  PROC DrawPart209()
    MoveL Offs(pOrigin,365.71,175.16,0.00),v40,z0,tPen\WObj:=wPaper;
    MoveL Offs(pOrigin,365.26,175.89,0.00),v40,z0,tPen\WObj:=wPaper;
    MoveL Offs(pOrigin,362.26,172.89,0.00),v40,z0,tPen\WObj:=wPaper;
    MoveL Offs(pOrigin,361.82,173.07,0.00),v40,z0,tPen\WObj:=wPaper;
    MoveL Offs(pOrigin,364.22,170.67,0.00),v40,z0,tPen\WObj:=wPaper;
    MoveL Offs(pOrigin,364.05,171.69,0.00),v40,z0,tPen\WObj:=wPaper;
    MoveL Offs(pOrigin,360.89,168.54,0.00),v40,z0,tPen\WObj:=wPaper;
    MoveL Offs(pOrigin,360.63,168.28,0.00),v40,z0,tPen\WObj:=wPaper;
    MoveL Offs(pOrigin,363.04,165.88,0.00),v40,z0,tPen\WObj:=wPaper;
    MoveL Offs(pOrigin,362.23,165.40,0.00),v40,z0,tPen\WObj:=wPaper;
    MoveL Offs(pOrigin,359.38,162.54,0.00),v40,z0,tPen\WObj:=wPaper;
    MoveL Offs(pOrigin,358.85,162.59,0.00),v40,z0,tPen\WObj:=wPaper;
    MoveL Offs(pOrigin,361.26,160.19,0.00),v40,z0,tPen\WObj:=wPaper;
    MoveL Offs(pOrigin,361.70,161.24,0.00),v40,z0,tPen\WObj:=wPaper;
    MoveL Offs(pOrigin,359.30,163.64,0.00),v40,z0,tPen\WObj:=wPaper;
    MoveL Offs(pOrigin,360.08,162.84,0.00),v40,z0,tPen\WObj:=wPaper;
    MoveL Offs(pOrigin,361.14,162.84,0.00),v40,z0,tPen\WObj:=wPaper;
    MoveL Offs(pOrigin,361.85,162.59,0.00),v40,z0,tPen\WObj:=wPaper;
    MoveL Offs(pOrigin,359.60,164.84,0.00),v40,z0,tPen\WObj:=wPaper;
    MoveL Offs(pOrigin,359.98,164.64,0.00),v40,z0,tPen\WObj:=wPaper;
    MoveL Offs(pOrigin,362.84,167.49,0.00),v40,z0,tPen\WObj:=wPaper;
    MoveL Offs(pOrigin,363.18,167.23,0.00),v40,z0,tPen\WObj:=wPaper;
    MoveL Offs(pOrigin,360.78,169.63,0.00),v40,z0,tPen\WObj:=wPaper;
    MoveL Offs(pOrigin,361.23,170.68,0.00),v40,z0,tPen\WObj:=wPaper;
    MoveL Offs(pOrigin,363.63,168.27,0.00),v40,fine,tPen\WObj:=wPaper;
    MoveL Offs(pOrigin,363.63,168.27,6.00),v60,z5,tPen\WObj:=wPaper;
    MoveL Offs(pOrigin,360.19,167.23,6.00),vTravel,z5,tPen\WObj:=wPaper;
    MoveL Offs(pOrigin,360.19,167.23,0.00),v60,z0,tPen\WObj:=wPaper;
    MoveL Offs(pOrigin,362.59,164.83,0.00),v40,fine,tPen\WObj:=wPaper;
    MoveL Offs(pOrigin,362.59,164.83,6.00),v60,z5,tPen\WObj:=wPaper;
    MoveL Offs(pOrigin,361.17,161.35,6.00),vTravel,z5,tPen\WObj:=wPaper;
    MoveL Offs(pOrigin,361.17,161.35,0.00),v60,z0,tPen\WObj:=wPaper;
    MoveL Offs(pOrigin,358.32,158.49,0.00),v40,z0,tPen\WObj:=wPaper;
    MoveL Offs(pOrigin,357.97,159.00,0.00),v40,z0,tPen\WObj:=wPaper;
    MoveL Offs(pOrigin,360.52,156.45,0.00),v40,fine,tPen\WObj:=wPaper;
    MoveL Offs(pOrigin,360.52,156.45,6.00),v60,z5,tPen\WObj:=wPaper;
    MoveL Offs(pOrigin,360.67,157.80,6.00),vTravel,z5,tPen\WObj:=wPaper;
    MoveL Offs(pOrigin,360.67,157.80,0.00),v60,z0,tPen\WObj:=wPaper;
    MoveL Offs(pOrigin,358.26,160.20,0.00),v40,fine,tPen\WObj:=wPaper;
    MoveL Offs(pOrigin,358.26,160.20,6.00),v60,z5,tPen\WObj:=wPaper;
    MoveL Offs(pOrigin,358.56,161.40,6.00),vTravel,z5,tPen\WObj:=wPaper;
    MoveL Offs(pOrigin,358.56,161.40,0.00),v60,z0,tPen\WObj:=wPaper;
    MoveL Offs(pOrigin,361.11,158.84,0.00),v40,fine,tPen\WObj:=wPaper;
    MoveL Offs(pOrigin,361.11,158.84,6.00),v60,z5,tPen\WObj:=wPaper;
    MoveL Offs(pOrigin,365.31,157.63,6.00),vTravel,z5,tPen\WObj:=wPaper;
    MoveL Offs(pOrigin,365.31,157.63,0.00),v60,z0,tPen\WObj:=wPaper;
    MoveL Offs(pOrigin,366.81,156.13,0.00),v40,z0,tPen\WObj:=wPaper;
    MoveL Offs(pOrigin,366.22,155.23,0.00),v40,z0,tPen\WObj:=wPaper;
    MoveL Offs(pOrigin,364.86,156.58,0.00),v40,z0,tPen\WObj:=wPaper;
    MoveL Offs(pOrigin,364.27,155.69,0.00),v40,z0,tPen\WObj:=wPaper;
    MoveL Offs(pOrigin,365.62,154.33,0.00),v40,z0,tPen\WObj:=wPaper;
    MoveL Offs(pOrigin,364.96,155.02,0.00),v40,z0,tPen\WObj:=wPaper;
    MoveL Offs(pOrigin,365.17,155.45,0.00),v40,z0,tPen\WObj:=wPaper;
    MoveL Offs(pOrigin,364.96,155.02,0.00),v40,fine,tPen\WObj:=wPaper;
    MoveL Offs(pOrigin,364.96,155.02,6.00),v60,z5,tPen\WObj:=wPaper;
    MoveL Offs(pOrigin,363.82,154.64,6.00),vTravel,z5,tPen\WObj:=wPaper;
    MoveL Offs(pOrigin,363.82,154.64,0.00),v60,z0,tPen\WObj:=wPaper;
    MoveL Offs(pOrigin,365.17,153.29,0.00),v40,z0,tPen\WObj:=wPaper;
    MoveL Offs(pOrigin,364.43,152.54,0.00),v40,z0,tPen\WObj:=wPaper;
    MoveL Offs(pOrigin,363.38,153.59,0.00),v40,z0,tPen\WObj:=wPaper;
    MoveL Offs(pOrigin,362.93,152.55,0.00),v40,z0,tPen\WObj:=wPaper;
    MoveL Offs(pOrigin,363.83,151.64,0.00),v40,fine,tPen\WObj:=wPaper;
    MoveL Offs(pOrigin,363.83,151.64,6.00),v60,z5,tPen\WObj:=wPaper;
    MoveL Offs(pOrigin,361.99,148.86,6.00),vTravel,z5,tPen\WObj:=wPaper;
    MoveL Offs(pOrigin,361.99,148.86,0.00),v60,z0,tPen\WObj:=wPaper;
    MoveL Offs(pOrigin,368.29,160.98,0.00),v40,z0,tPen\WObj:=wPaper;
    MoveL Offs(pOrigin,376.86,174.36,0.00),v40,z0,tPen\WObj:=wPaper;
    MoveL Offs(pOrigin,377.69,175.12,0.00),v40,z0,tPen\WObj:=wPaper;
    MoveL Offs(pOrigin,382.35,170.46,0.00),v40,fine,tPen\WObj:=wPaper;
    MoveL Offs(pOrigin,382.35,170.46,6.00),v60,z5,tPen\WObj:=wPaper;
    MoveL Offs(pOrigin,382.34,171.96,6.00),vTravel,z5,tPen\WObj:=wPaper;
    MoveL Offs(pOrigin,382.34,171.96,0.00),v60,z0,tPen\WObj:=wPaper;
    MoveL Offs(pOrigin,377.24,177.07,0.00),v40,fine,tPen\WObj:=wPaper;
    MoveL Offs(pOrigin,377.24,177.07,6.00),v60,z5,tPen\WObj:=wPaper;
    MoveL Offs(pOrigin,376.78,179.02,6.00),vTravel,z5,tPen\WObj:=wPaper;
    MoveL Offs(pOrigin,376.78,179.02,0.00),v60,z0,tPen\WObj:=wPaper;
    MoveL Offs(pOrigin,381.74,174.06,0.00),v40,fine,tPen\WObj:=wPaper;
    MoveL Offs(pOrigin,381.74,174.06,6.00),v60,z5,tPen\WObj:=wPaper;
    MoveL Offs(pOrigin,378.75,172.57,6.00),vTravel,z5,tPen\WObj:=wPaper;
    MoveL Offs(pOrigin,378.75,172.57,0.00),v60,z0,tPen\WObj:=wPaper;
    MoveL Offs(pOrigin,382.35,168.96,0.00),v40,fine,tPen\WObj:=wPaper;
    MoveL Offs(pOrigin,382.35,168.96,6.00),v60,z5,tPen\WObj:=wPaper;
    MoveL Offs(pOrigin,380.69,164.95,6.00),vTravel,z5,tPen\WObj:=wPaper;
    MoveL Offs(pOrigin,380.69,164.95,0.00),v60,z0,tPen\WObj:=wPaper;
    MoveL Offs(pOrigin,377.92,164.95,0.00),v40,z0,tPen\WObj:=wPaper;
    MoveL Offs(pOrigin,376.97,165.39,0.00),v40,z0,tPen\WObj:=wPaper;
    MoveL Offs(pOrigin,384.03,158.32,0.00),v40,fine,tPen\WObj:=wPaper;
    MoveL Offs(pOrigin,384.03,158.32,6.00),v60,z5,tPen\WObj:=wPaper;
    MoveL Offs(pOrigin,385.24,155.62,6.00),vTravel,z5,tPen\WObj:=wPaper;
    MoveL Offs(pOrigin,385.24,155.62,0.00),v60,z0,tPen\WObj:=wPaper;
    MoveL Offs(pOrigin,376.38,164.49,0.00),v40,z0,tPen\WObj:=wPaper;
    MoveL Offs(pOrigin,376.86,163.95,0.00),v40,z0,tPen\WObj:=wPaper;
    MoveL Offs(pOrigin,377.29,164.38,0.00),v40,z0,tPen\WObj:=wPaper;
    MoveL Offs(pOrigin,376.86,163.95,0.00),v40,z0,tPen\WObj:=wPaper;
    MoveL Offs(pOrigin,376.23,163.10,0.00),v40,z0,tPen\WObj:=wPaper;
    MoveL Offs(pOrigin,376.65,163.52,0.00),v40,z0,tPen\WObj:=wPaper;
    MoveL Offs(pOrigin,376.23,163.10,0.00),v40,fine,tPen\WObj:=wPaper;
    MoveL Offs(pOrigin,376.23,163.10,6.00),v60,z5,tPen\WObj:=wPaper;
    MoveL Offs(pOrigin,372.33,165.55,6.00),vTravel,z5,tPen\WObj:=wPaper;
    MoveL Offs(pOrigin,372.33,165.55,0.00),v60,z0,tPen\WObj:=wPaper;
    MoveL Offs(pOrigin,370.67,167.20,0.00),v40,z0,tPen\WObj:=wPaper;
    MoveL Offs(pOrigin,371.42,167.95,0.00),v40,z0,tPen\WObj:=wPaper;
    MoveL Offs(pOrigin,372.77,166.60,0.00),v40,z0,tPen\WObj:=wPaper;
    MoveL Offs(pOrigin,373.52,167.34,0.00),v40,z0,tPen\WObj:=wPaper;
    MoveL Offs(pOrigin,372.02,168.85,0.00),v40,z0,tPen\WObj:=wPaper;
    MoveL Offs(pOrigin,372.61,169.74,0.00),v40,z0,tPen\WObj:=wPaper;
    MoveL Offs(pOrigin,373.97,168.39,0.00),v40,z0,tPen\WObj:=wPaper;
    MoveL Offs(pOrigin,374.56,169.29,0.00),v40,z0,tPen\WObj:=wPaper;
    MoveL Offs(pOrigin,373.21,170.64,0.00),v40,z0,tPen\WObj:=wPaper;
    MoveL Offs(pOrigin,373.96,171.39,0.00),v40,z0,tPen\WObj:=wPaper;
    MoveL Offs(pOrigin,375.16,170.18,0.00),v40,z0,tPen\WObj:=wPaper;
    MoveL Offs(pOrigin,375.76,171.08,0.00),v40,z0,tPen\WObj:=wPaper;
    MoveL Offs(pOrigin,374.55,172.28,0.00),v40,z0,tPen\WObj:=wPaper;
    MoveL Offs(pOrigin,375.30,173.03,0.00),v40,z0,tPen\WObj:=wPaper;
    MoveL Offs(pOrigin,376.20,172.13,0.00),v40,fine,tPen\WObj:=wPaper;
    MoveL Offs(pOrigin,376.20,172.13,6.00),v60,z5,tPen\WObj:=wPaper;
    MoveL Offs(pOrigin,373.67,169.69,6.00),vTravel,z5,tPen\WObj:=wPaper;
    MoveL Offs(pOrigin,373.67,169.69,0.00),v60,z0,tPen\WObj:=wPaper;
    MoveL Offs(pOrigin,374.10,170.32,0.00),v40,z0,tPen\WObj:=wPaper;
    MoveL Offs(pOrigin,373.67,169.69,0.00),v40,fine,tPen\WObj:=wPaper;
  ENDPROC

  PROC DrawPart210()
    MoveL Offs(pOrigin,373.67,169.69,6.00),v60,z5,tPen\WObj:=wPaper;
    MoveL Offs(pOrigin,371.82,166.02,6.00),vTravel,z5,tPen\WObj:=wPaper;
    MoveL Offs(pOrigin,371.82,166.02,0.00),v60,z0,tPen\WObj:=wPaper;
    MoveL Offs(pOrigin,369.12,163.32,0.00),v40,z0,tPen\WObj:=wPaper;
    MoveL Offs(pOrigin,368.44,163.46,0.00),v40,z0,tPen\WObj:=wPaper;
    MoveL Offs(pOrigin,370.24,161.66,0.00),v40,z0,tPen\WObj:=wPaper;
    MoveL Offs(pOrigin,369.86,162.57,0.00),v40,z0,tPen\WObj:=wPaper;
    MoveL Offs(pOrigin,367.46,160.17,0.00),v40,z0,tPen\WObj:=wPaper;
    MoveL Offs(pOrigin,366.95,160.47,0.00),v40,z0,tPen\WObj:=wPaper;
    MoveL Offs(pOrigin,368.45,158.97,0.00),v40,z0,tPen\WObj:=wPaper;
    MoveL Offs(pOrigin,367.86,158.07,0.00),v40,z0,tPen\WObj:=wPaper;
    MoveL Offs(pOrigin,366.35,159.58,0.00),v40,z0,tPen\WObj:=wPaper;
    MoveL Offs(pOrigin,365.91,158.53,0.00),v40,z0,tPen\WObj:=wPaper;
    MoveL Offs(pOrigin,367.26,157.18,0.00),v40,z0,tPen\WObj:=wPaper;
    MoveL Offs(pOrigin,366.45,157.79,0.00),v40,z0,tPen\WObj:=wPaper;
    MoveL Offs(pOrigin,366.66,158.21,0.00),v40,z0,tPen\WObj:=wPaper;
    MoveL Offs(pOrigin,366.45,157.79,0.00),v40,fine,tPen\WObj:=wPaper;
    MoveL Offs(pOrigin,366.45,157.79,6.00),v60,z5,tPen\WObj:=wPaper;
    MoveL Offs(pOrigin,368.90,160.02,6.00),vTravel,z5,tPen\WObj:=wPaper;
    MoveL Offs(pOrigin,368.90,160.02,0.00),v60,z0,tPen\WObj:=wPaper;
    MoveL Offs(pOrigin,367.40,161.52,0.00),v40,z0,tPen\WObj:=wPaper;
    MoveL Offs(pOrigin,367.99,162.42,0.00),v40,z0,tPen\WObj:=wPaper;
    MoveL Offs(pOrigin,369.50,160.91,0.00),v40,fine,tPen\WObj:=wPaper;
    MoveL Offs(pOrigin,369.50,160.91,6.00),v60,z5,tPen\WObj:=wPaper;
    MoveL Offs(pOrigin,370.69,162.71,6.00),vTravel,z5,tPen\WObj:=wPaper;
    MoveL Offs(pOrigin,370.69,162.71,0.00),v60,z0,tPen\WObj:=wPaper;
    MoveL Offs(pOrigin,369.04,164.36,0.00),v40,z0,tPen\WObj:=wPaper;
    MoveL Offs(pOrigin,369.48,165.41,0.00),v40,z0,tPen\WObj:=wPaper;
    MoveL Offs(pOrigin,371.28,163.60,0.00),v40,z0,tPen\WObj:=wPaper;
    MoveL Offs(pOrigin,371.73,164.65,0.00),v40,z0,tPen\WObj:=wPaper;
    MoveL Offs(pOrigin,370.23,166.15,0.00),v40,fine,tPen\WObj:=wPaper;
    MoveL Offs(pOrigin,370.23,166.15,6.00),v60,z5,tPen\WObj:=wPaper;
    MoveL Offs(pOrigin,365.85,176.50,6.00),vTravel,z5,tPen\WObj:=wPaper;
    MoveL Offs(pOrigin,365.85,176.50,0.00),v60,z0,tPen\WObj:=wPaper;
    MoveL Offs(pOrigin,363.75,178.61,0.00),v40,fine,tPen\WObj:=wPaper;
    MoveL Offs(pOrigin,363.75,178.61,6.00),v60,z5,tPen\WObj:=wPaper;
    MoveL Offs(pOrigin,364.64,180.70,6.00),vTravel,z5,tPen\WObj:=wPaper;
    MoveL Offs(pOrigin,364.64,180.70,0.00),v60,z0,tPen\WObj:=wPaper;
    MoveL Offs(pOrigin,366.74,178.60,0.00),v40,fine,tPen\WObj:=wPaper;
    MoveL Offs(pOrigin,366.74,178.60,6.00),v60,z5,tPen\WObj:=wPaper;
    MoveL Offs(pOrigin,367.49,180.84,6.00),vTravel,z5,tPen\WObj:=wPaper;
    MoveL Offs(pOrigin,367.49,180.84,0.00),v60,z0,tPen\WObj:=wPaper;
    MoveL Offs(pOrigin,365.38,182.95,0.00),v40,z0,tPen\WObj:=wPaper;
    MoveL Offs(pOrigin,365.83,183.99,0.00),v40,z0,tPen\WObj:=wPaper;
    MoveL Offs(pOrigin,367.93,181.89,0.00),v40,fine,tPen\WObj:=wPaper;
    MoveL Offs(pOrigin,367.93,181.89,6.00),v60,z5,tPen\WObj:=wPaper;
    MoveL Offs(pOrigin,371.06,187.72,6.00),vTravel,z5,tPen\WObj:=wPaper;
    MoveL Offs(pOrigin,371.06,187.72,0.00),v60,z0,tPen\WObj:=wPaper;
    MoveL Offs(pOrigin,365.50,193.28,0.00),v40,z0,tPen\WObj:=wPaper;
    MoveL Offs(pOrigin,365.76,192.82,0.00),v40,z0,tPen\WObj:=wPaper;
    MoveL Offs(pOrigin,364.26,191.32,0.00),v40,fine,tPen\WObj:=wPaper;
    MoveL Offs(pOrigin,364.26,191.32,6.00),v60,z5,tPen\WObj:=wPaper;
    MoveL Offs(pOrigin,365.46,191.02,6.00),vTravel,z5,tPen\WObj:=wPaper;
    MoveL Offs(pOrigin,365.46,191.02,0.00),v60,z0,tPen\WObj:=wPaper;
    MoveL Offs(pOrigin,366.81,192.37,0.00),v40,z0,tPen\WObj:=wPaper;
    MoveL Offs(pOrigin,367.60,192.68,0.00),v40,z0,tPen\WObj:=wPaper;
    MoveL Offs(pOrigin,372.26,188.02,0.00),v40,z0,tPen\WObj:=wPaper;
    MoveL Offs(pOrigin,372.19,188.79,0.00),v40,z0,tPen\WObj:=wPaper;
    MoveL Offs(pOrigin,374.29,190.90,0.00),v40,z0,tPen\WObj:=wPaper;
    MoveL Offs(pOrigin,373.89,190.30,0.00),v40,z0,tPen\WObj:=wPaper;
    MoveL Offs(pOrigin,369.00,190.30,0.00),v40,z0,tPen\WObj:=wPaper;
    MoveL Offs(pOrigin,367.85,190.43,0.00),v40,z0,tPen\WObj:=wPaper;
    MoveL Offs(pOrigin,369.20,191.78,0.00),v40,z0,tPen\WObj:=wPaper;
    MoveL Offs(pOrigin,368.36,191.35,0.00),v40,z0,tPen\WObj:=wPaper;
    MoveL Offs(pOrigin,366.02,191.35,0.00),v40,z0,tPen\WObj:=wPaper;
    MoveL Offs(pOrigin,366.50,190.57,0.00),v40,z0,tPen\WObj:=wPaper;
    MoveL Offs(pOrigin,368.01,192.08,0.00),v40,fine,tPen\WObj:=wPaper;
    MoveL Offs(pOrigin,368.01,192.08,6.00),v60,z5,tPen\WObj:=wPaper;
    MoveL Offs(pOrigin,365.51,190.29,6.00),vTravel,z5,tPen\WObj:=wPaper;
    MoveL Offs(pOrigin,365.51,190.29,0.00),v60,z0,tPen\WObj:=wPaper;
    MoveL Offs(pOrigin,361.45,194.34,0.00),v40,z0,tPen\WObj:=wPaper;
    MoveL Offs(pOrigin,362.17,193.71,0.00),v40,z0,tPen\WObj:=wPaper;
    MoveL Offs(pOrigin,360.67,192.20,0.00),v40,z0,tPen\WObj:=wPaper;
    MoveL Offs(pOrigin,361.46,191.35,0.00),v40,z0,tPen\WObj:=wPaper;
    MoveL Offs(pOrigin,357.41,195.40,0.00),v40,z0,tPen\WObj:=wPaper;
    MoveL Offs(pOrigin,356.33,195.34,0.00),v40,z0,tPen\WObj:=wPaper;
    MoveL Offs(pOrigin,354.68,193.68,0.00),v40,fine,tPen\WObj:=wPaper;
    MoveL Offs(pOrigin,354.68,193.68,6.00),v60,z5,tPen\WObj:=wPaper;
    MoveL Offs(pOrigin,353.37,193.47,6.00),vTravel,z5,tPen\WObj:=wPaper;
    MoveL Offs(pOrigin,353.37,193.47,0.00),v60,z0,tPen\WObj:=wPaper;
    MoveL Offs(pOrigin,349.01,197.83,0.00),v40,fine,tPen\WObj:=wPaper;
    MoveL Offs(pOrigin,349.01,197.83,6.00),v60,z5,tPen\WObj:=wPaper;
    MoveL Offs(pOrigin,346.91,198.43,6.00),vTravel,z5,tPen\WObj:=wPaper;
    MoveL Offs(pOrigin,346.91,198.43,0.00),v60,z0,tPen\WObj:=wPaper;
    MoveL Offs(pOrigin,351.27,194.08,0.00),v40,z0,tPen\WObj:=wPaper;
    MoveL Offs(pOrigin,351.24,194.72,0.00),v40,z0,tPen\WObj:=wPaper;
    MoveL Offs(pOrigin,352.59,196.07,0.00),v40,z0,tPen\WObj:=wPaper;
    MoveL Offs(pOrigin,352.85,195.58,0.00),v40,z0,tPen\WObj:=wPaper;
    MoveL Offs(pOrigin,349.88,195.58,0.00),v40,z0,tPen\WObj:=wPaper;
    MoveL Offs(pOrigin,350.04,195.02,0.00),v40,z0,tPen\WObj:=wPaper;
    MoveL Offs(pOrigin,351.54,196.52,0.00),v40,fine,tPen\WObj:=wPaper;
    MoveL Offs(pOrigin,351.54,196.52,6.00),v60,z5,tPen\WObj:=wPaper;
    MoveL Offs(pOrigin,353.21,196.62,6.00),vTravel,z5,tPen\WObj:=wPaper;
    MoveL Offs(pOrigin,353.21,196.62,0.00),v60,z0,tPen\WObj:=wPaper;
    MoveL Offs(pOrigin,357.41,192.41,0.00),v40,z0,tPen\WObj:=wPaper;
    MoveL Offs(pOrigin,357.07,193.09,0.00),v40,z0,tPen\WObj:=wPaper;
    MoveL Offs(pOrigin,358.58,194.59,0.00),v40,fine,tPen\WObj:=wPaper;
    MoveL Offs(pOrigin,358.58,194.59,6.00),v60,z5,tPen\WObj:=wPaper;
    MoveL Offs(pOrigin,353.94,195.93,6.00),vTravel,z5,tPen\WObj:=wPaper;
    MoveL Offs(pOrigin,353.94,195.93,0.00),v60,z0,tPen\WObj:=wPaper;
    MoveL Offs(pOrigin,352.28,194.28,0.00),v40,fine,tPen\WObj:=wPaper;
    MoveL Offs(pOrigin,352.28,194.28,6.00),v60,z5,tPen\WObj:=wPaper;
    MoveL Offs(pOrigin,341.59,181.80,6.00),vTravel,z5,tPen\WObj:=wPaper;
    MoveL Offs(pOrigin,341.59,181.80,0.00),v60,z0,tPen\WObj:=wPaper;
    MoveL Offs(pOrigin,334.15,175.85,0.00),v40,z0,tPen\WObj:=wPaper;
    MoveL Offs(pOrigin,330.33,172.02,0.00),v40,z0,tPen\WObj:=wPaper;
    MoveL Offs(pOrigin,323.74,164.16,0.00),v40,z0,tPen\WObj:=wPaper;
    MoveL Offs(pOrigin,315.38,151.84,0.00),v40,z0,tPen\WObj:=wPaper;
    MoveL Offs(pOrigin,309.85,141.64,0.00),v40,z0,tPen\WObj:=wPaper;
    MoveL Offs(pOrigin,309.08,139.51,0.00),v40,fine,tPen\WObj:=wPaper;
    MoveL Offs(pOrigin,309.08,139.51,6.00),v60,z5,tPen\WObj:=wPaper;
    MoveL Offs(pOrigin,304.61,138.55,6.00),vTravel,z5,tPen\WObj:=wPaper;
    MoveL Offs(pOrigin,304.61,138.55,0.00),v60,z0,tPen\WObj:=wPaper;
    MoveL Offs(pOrigin,303.55,138.55,0.00),v40,z0,tPen\WObj:=wPaper;
    MoveL Offs(pOrigin,303.12,137.50,0.00),v40,z0,tPen\WObj:=wPaper;
    MoveL Offs(pOrigin,304.19,137.50,0.00),v40,z0,tPen\WObj:=wPaper;
    MoveL Offs(pOrigin,305.15,137.14,0.00),v40,z0,tPen\WObj:=wPaper;
    MoveL Offs(pOrigin,302.75,139.55,0.00),v40,fine,tPen\WObj:=wPaper;
    MoveL Offs(pOrigin,302.75,139.55,6.00),v60,z5,tPen\WObj:=wPaper;
    MoveL Offs(pOrigin,299.34,129.52,6.00),vTravel,z5,tPen\WObj:=wPaper;
  ENDPROC

  PROC DrawPart211()
    MoveL Offs(pOrigin,299.34,129.52,0.00),v60,z0,tPen\WObj:=wPaper;
    MoveL Offs(pOrigin,302.04,126.82,0.00),v40,fine,tPen\WObj:=wPaper;
    MoveL Offs(pOrigin,302.04,126.82,6.00),v60,z5,tPen\WObj:=wPaper;
    MoveL Offs(pOrigin,301.15,124.72,6.00),vTravel,z5,tPen\WObj:=wPaper;
    MoveL Offs(pOrigin,301.15,124.72,0.00),v60,z0,tPen\WObj:=wPaper;
    MoveL Offs(pOrigin,298.74,127.13,0.00),v40,fine,tPen\WObj:=wPaper;
    MoveL Offs(pOrigin,298.74,127.13,6.00),v60,z5,tPen\WObj:=wPaper;
    MoveL Offs(pOrigin,302.36,119.03,6.00),vTravel,z5,tPen\WObj:=wPaper;
    MoveL Offs(pOrigin,302.36,119.03,0.00),v60,z0,tPen\WObj:=wPaper;
    MoveL Offs(pOrigin,305.82,115.57,0.00),v40,z0,tPen\WObj:=wPaper;
    MoveL Offs(pOrigin,306.87,116.02,0.00),v40,z0,tPen\WObj:=wPaper;
    MoveL Offs(pOrigin,303.41,119.47,0.00),v40,z0,tPen\WObj:=wPaper;
    MoveL Offs(pOrigin,304.12,119.23,0.00),v40,z0,tPen\WObj:=wPaper;
    MoveL Offs(pOrigin,301.71,116.82,0.00),v40,fine,tPen\WObj:=wPaper;
    MoveL Offs(pOrigin,301.71,116.82,6.00),v60,z5,tPen\WObj:=wPaper;
    MoveL Offs(pOrigin,304.11,117.73,6.00),vTravel,z5,tPen\WObj:=wPaper;
    MoveL Offs(pOrigin,304.11,117.73,0.00),v60,z0,tPen\WObj:=wPaper;
    MoveL Offs(pOrigin,306.37,119.98,0.00),v40,z0,tPen\WObj:=wPaper;
    MoveL Offs(pOrigin,305.81,120.06,0.00),v40,z0,tPen\WObj:=wPaper;
    MoveL Offs(pOrigin,309.41,116.46,0.00),v40,z0,tPen\WObj:=wPaper;
    MoveL Offs(pOrigin,310.46,116.90,0.00),v40,z0,tPen\WObj:=wPaper;
    MoveL Offs(pOrigin,307.00,120.36,0.00),v40,z0,tPen\WObj:=wPaper;
    MoveL Offs(pOrigin,308.05,120.81,0.00),v40,z0,tPen\WObj:=wPaper;
    MoveL Offs(pOrigin,311.81,117.05,0.00),v40,fine,tPen\WObj:=wPaper;
    MoveL Offs(pOrigin,311.81,117.05,6.00),v60,z5,tPen\WObj:=wPaper;
    MoveL Offs(pOrigin,313.00,117.35,6.00),vTravel,z5,tPen\WObj:=wPaper;
    MoveL Offs(pOrigin,313.00,117.35,0.00),v60,z0,tPen\WObj:=wPaper;
    MoveL Offs(pOrigin,309.40,120.95,0.00),v40,z0,tPen\WObj:=wPaper;
    MoveL Offs(pOrigin,308.47,120.59,0.00),v40,z0,tPen\WObj:=wPaper;
    MoveL Offs(pOrigin,306.06,118.19,0.00),v40,fine,tPen\WObj:=wPaper;
    MoveL Offs(pOrigin,306.06,118.19,6.00),v60,z5,tPen\WObj:=wPaper;
    MoveL Offs(pOrigin,304.61,119.77,6.00),vTravel,z5,tPen\WObj:=wPaper;
    MoveL Offs(pOrigin,304.61,119.77,0.00),v60,z0,tPen\WObj:=wPaper;
    MoveL Offs(pOrigin,308.22,116.16,0.00),v40,fine,tPen\WObj:=wPaper;
    MoveL Offs(pOrigin,308.22,116.16,6.00),v60,z5,tPen\WObj:=wPaper;
    MoveL Offs(pOrigin,308.16,118.79,6.00),vTravel,z5,tPen\WObj:=wPaper;
    MoveL Offs(pOrigin,308.16,118.79,0.00),v60,z0,tPen\WObj:=wPaper;
    MoveL Offs(pOrigin,310.42,121.05,0.00),v40,z0,tPen\WObj:=wPaper;
    MoveL Offs(pOrigin,310.45,121.40,0.00),v40,z0,tPen\WObj:=wPaper;
    MoveL Offs(pOrigin,314.20,117.64,0.00),v40,fine,tPen\WObj:=wPaper;
    MoveL Offs(pOrigin,314.20,117.64,6.00),v60,z5,tPen\WObj:=wPaper;
    MoveL Offs(pOrigin,315.40,117.94,6.00),vTravel,z5,tPen\WObj:=wPaper;
    MoveL Offs(pOrigin,315.40,117.94,0.00),v60,z0,tPen\WObj:=wPaper;
    MoveL Offs(pOrigin,311.79,121.54,0.00),v40,z0,tPen\WObj:=wPaper;
    MoveL Offs(pOrigin,312.51,121.65,0.00),v40,z0,tPen\WObj:=wPaper;
    MoveL Offs(pOrigin,310.11,119.25,0.00),v40,fine,tPen\WObj:=wPaper;
    MoveL Offs(pOrigin,310.11,119.25,6.00),v60,z5,tPen\WObj:=wPaper;
    MoveL Offs(pOrigin,312.84,121.99,6.00),vTravel,z5,tPen\WObj:=wPaper;
    MoveL Offs(pOrigin,312.84,121.99,0.00),v60,z0,tPen\WObj:=wPaper;
    MoveL Offs(pOrigin,316.45,118.38,0.00),v40,fine,tPen\WObj:=wPaper;
    MoveL Offs(pOrigin,316.45,118.38,6.00),v60,z5,tPen\WObj:=wPaper;
    MoveL Offs(pOrigin,356.89,119.54,6.00),vTravel,z5,tPen\WObj:=wPaper;
    MoveL Offs(pOrigin,356.89,119.54,0.00),v60,z0,tPen\WObj:=wPaper;
    MoveL Offs(pOrigin,357.31,119.96,0.00),v40,z0,tPen\WObj:=wPaper;
    MoveL Offs(pOrigin,356.89,119.54,0.00),v40,fine,tPen\WObj:=wPaper;
    MoveL Offs(pOrigin,356.89,119.54,6.00),v60,z5,tPen\WObj:=wPaper;
    MoveL Offs(pOrigin,365.73,118.38,6.00),vTravel,z5,tPen\WObj:=wPaper;
    MoveL Offs(pOrigin,365.73,118.38,0.00),v60,z0,tPen\WObj:=wPaper;
    MoveL Offs(pOrigin,367.23,116.88,0.00),v40,z0,tPen\WObj:=wPaper;
    MoveL Offs(pOrigin,368.13,117.48,0.00),v40,z0,tPen\WObj:=wPaper;
    MoveL Offs(pOrigin,367.08,118.53,0.00),v40,fine,tPen\WObj:=wPaper;
    MoveL Offs(pOrigin,367.08,118.53,6.00),v60,z5,tPen\WObj:=wPaper;
    MoveL Offs(pOrigin,366.19,114.94,6.00),vTravel,z5,tPen\WObj:=wPaper;
    MoveL Offs(pOrigin,366.19,114.94,0.00),v60,z0,tPen\WObj:=wPaper;
    MoveL Offs(pOrigin,367.84,113.28,0.00),v40,fine,tPen\WObj:=wPaper;
    MoveL Offs(pOrigin,367.84,113.28,6.00),v60,z5,tPen\WObj:=wPaper;
    MoveL Offs(pOrigin,368.90,109.24,6.00),vTravel,z5,tPen\WObj:=wPaper;
    MoveL Offs(pOrigin,368.90,109.24,0.00),v60,z0,tPen\WObj:=wPaper;
    MoveL Offs(pOrigin,371.01,107.13,0.00),v40,z0,tPen\WObj:=wPaper;
    MoveL Offs(pOrigin,370.44,107.90,0.00),v40,z0,tPen\WObj:=wPaper;
    MoveL Offs(pOrigin,371.80,109.25,0.00),v40,z0,tPen\WObj:=wPaper;
    MoveL Offs(pOrigin,371.60,109.53,0.00),v40,z0,tPen\WObj:=wPaper;
    MoveL Offs(pOrigin,373.85,107.27,0.00),v40,z0,tPen\WObj:=wPaper;
    MoveL Offs(pOrigin,373.59,108.06,0.00),v40,z0,tPen\WObj:=wPaper;
    MoveL Offs(pOrigin,374.79,109.26,0.00),v40,z0,tPen\WObj:=wPaper;
    MoveL Offs(pOrigin,374.45,109.67,0.00),v40,z0,tPen\WObj:=wPaper;
    MoveL Offs(pOrigin,376.85,107.26,0.00),v40,fine,tPen\WObj:=wPaper;
    MoveL Offs(pOrigin,376.85,107.26,6.00),v60,z5,tPen\WObj:=wPaper;
    MoveL Offs(pOrigin,378.08,108.07,6.00),vTravel,z5,tPen\WObj:=wPaper;
    MoveL Offs(pOrigin,378.08,108.07,0.00),v60,z0,tPen\WObj:=wPaper;
    MoveL Offs(pOrigin,378.99,108.97,0.00),v40,z0,tPen\WObj:=wPaper;
    MoveL Offs(pOrigin,379.09,109.50,0.00),v40,z0,tPen\WObj:=wPaper;
    MoveL Offs(pOrigin,381.80,106.80,0.00),v40,fine,tPen\WObj:=wPaper;
    MoveL Offs(pOrigin,381.80,106.80,6.00),v60,z5,tPen\WObj:=wPaper;
    MoveL Offs(pOrigin,380.93,107.93,6.00),vTravel,z5,tPen\WObj:=wPaper;
    MoveL Offs(pOrigin,380.93,107.93,0.00),v60,z0,tPen\WObj:=wPaper;
    MoveL Offs(pOrigin,381.68,108.68,0.00),v40,z0,tPen\WObj:=wPaper;
    MoveL Offs(pOrigin,380.89,109.20,0.00),v40,z0,tPen\WObj:=wPaper;
    MoveL Offs(pOrigin,383.44,106.64,0.00),v40,fine,tPen\WObj:=wPaper;
    MoveL Offs(pOrigin,383.44,106.64,6.00),v60,z5,tPen\WObj:=wPaper;
    MoveL Offs(pOrigin,383.15,105.45,6.00),vTravel,z5,tPen\WObj:=wPaper;
    MoveL Offs(pOrigin,383.15,105.45,0.00),v60,z0,tPen\WObj:=wPaper;
    MoveL Offs(pOrigin,387.05,101.54,0.00),v40,z0,tPen\WObj:=wPaper;
    MoveL Offs(pOrigin,387.36,102.41,0.00),v40,z0,tPen\WObj:=wPaper;
    MoveL Offs(pOrigin,388.56,103.61,0.00),v40,z0,tPen\WObj:=wPaper;
    MoveL Offs(pOrigin,389.14,103.93,0.00),v40,z0,tPen\WObj:=wPaper;
    MoveL Offs(pOrigin,394.10,98.97,0.00),v40,z0,tPen\WObj:=wPaper;
    MoveL Offs(pOrigin,393.94,100.03,0.00),v40,z0,tPen\WObj:=wPaper;
    MoveL Offs(pOrigin,394.99,101.08,0.00),v40,z0,tPen\WObj:=wPaper;
    MoveL Offs(pOrigin,393.94,101.53,0.00),v40,z0,tPen\WObj:=wPaper;
    MoveL Offs(pOrigin,392.74,100.33,0.00),v40,z0,tPen\WObj:=wPaper;
    MoveL Offs(pOrigin,393.44,100.84,0.00),v40,z0,tPen\WObj:=wPaper;
    MoveL Offs(pOrigin,384.51,103.39,0.00),v40,z0,tPen\WObj:=wPaper;
    MoveL Offs(pOrigin,379.20,104.24,0.00),v40,z0,tPen\WObj:=wPaper;
    MoveL Offs(pOrigin,371.55,104.24,0.00),v40,z0,tPen\WObj:=wPaper;
    MoveL Offs(pOrigin,365.39,102.75,0.00),v40,fine,tPen\WObj:=wPaper;
    MoveL Offs(pOrigin,365.39,102.75,6.00),v60,z5,tPen\WObj:=wPaper;
    MoveL Offs(pOrigin,366.07,104.60,6.00),vTravel,z5,tPen\WObj:=wPaper;
    MoveL Offs(pOrigin,366.07,104.60,0.00),v60,z0,tPen\WObj:=wPaper;
    MoveL Offs(pOrigin,368.18,102.50,0.00),v40,z0,tPen\WObj:=wPaper;
    MoveL Offs(pOrigin,368.93,103.40,0.00),v40,z0,tPen\WObj:=wPaper;
    MoveL Offs(pOrigin,370.89,105.35,0.00),v40,z0,tPen\WObj:=wPaper;
    MoveL Offs(pOrigin,371.01,105.63,0.00),v40,z0,tPen\WObj:=wPaper;
    MoveL Offs(pOrigin,373.42,103.23,0.00),v40,z0,tPen\WObj:=wPaper;
    MoveL Offs(pOrigin,374.03,104.01,0.00),v40,z0,tPen\WObj:=wPaper;
    MoveL Offs(pOrigin,375.83,105.82,0.00),v40,z0,tPen\WObj:=wPaper;
    MoveL Offs(pOrigin,375.06,106.07,0.00),v40,z0,tPen\WObj:=wPaper;
    MoveL Offs(pOrigin,377.91,103.22,0.00),v40,z0,tPen\WObj:=wPaper;
    MoveL Offs(pOrigin,378.37,103.88,0.00),v40,z0,tPen\WObj:=wPaper;
    MoveL Offs(pOrigin,379.87,105.38,0.00),v40,z0,tPen\WObj:=wPaper;
  ENDPROC

  PROC DrawPart212()
    MoveL Offs(pOrigin,379.70,105.91,0.00),v40,z0,tPen\WObj:=wPaper;
    MoveL Offs(pOrigin,383.01,102.60,0.00),v40,z0,tPen\WObj:=wPaper;
    MoveL Offs(pOrigin,383.76,103.29,0.00),v40,z0,tPen\WObj:=wPaper;
    MoveL Offs(pOrigin,385.12,104.65,0.00),v40,fine,tPen\WObj:=wPaper;
    MoveL Offs(pOrigin,385.12,104.65,6.00),v60,z5,tPen\WObj:=wPaper;
    MoveL Offs(pOrigin,383.77,104.79,6.00),vTravel,z5,tPen\WObj:=wPaper;
    MoveL Offs(pOrigin,383.77,104.79,0.00),v60,z0,tPen\WObj:=wPaper;
    MoveL Offs(pOrigin,382.41,103.44,0.00),v40,fine,tPen\WObj:=wPaper;
    MoveL Offs(pOrigin,382.41,103.44,6.00),v60,z5,tPen\WObj:=wPaper;
    MoveL Offs(pOrigin,381.22,103.74,6.00),vTravel,z5,tPen\WObj:=wPaper;
    MoveL Offs(pOrigin,381.22,103.74,0.00),v60,z0,tPen\WObj:=wPaper;
    MoveL Offs(pOrigin,382.57,105.09,0.00),v40,fine,tPen\WObj:=wPaper;
    MoveL Offs(pOrigin,382.57,105.09,6.00),v60,z5,tPen\WObj:=wPaper;
    MoveL Offs(pOrigin,381.36,102.76,6.00),vTravel,z5,tPen\WObj:=wPaper;
    MoveL Offs(pOrigin,381.36,102.76,0.00),v60,z0,tPen\WObj:=wPaper;
    MoveL Offs(pOrigin,378.05,106.06,0.00),v40,z0,tPen\WObj:=wPaper;
    MoveL Offs(pOrigin,378.68,105.68,0.00),v40,z0,tPen\WObj:=wPaper;
    MoveL Offs(pOrigin,377.02,104.02,0.00),v40,z0,tPen\WObj:=wPaper;
    MoveL Offs(pOrigin,377.29,104.76,0.00),v40,z0,tPen\WObj:=wPaper;
    MoveL Offs(pOrigin,373.67,104.76,0.00),v40,fine,tPen\WObj:=wPaper;
    MoveL Offs(pOrigin,373.67,104.76,6.00),v60,z5,tPen\WObj:=wPaper;
    MoveL Offs(pOrigin,374.33,105.81,6.00),vTravel,z5,tPen\WObj:=wPaper;
    MoveL Offs(pOrigin,374.33,105.81,0.00),v60,z0,tPen\WObj:=wPaper;
    MoveL Offs(pOrigin,372.38,103.86,0.00),v40,z0,tPen\WObj:=wPaper;
    MoveL Offs(pOrigin,371.92,103.23,0.00),v40,z0,tPen\WObj:=wPaper;
    MoveL Offs(pOrigin,369.67,105.49,0.00),v40,fine,tPen\WObj:=wPaper;
    MoveL Offs(pOrigin,369.67,105.49,6.00),v60,z5,tPen\WObj:=wPaper;
    MoveL Offs(pOrigin,369.51,107.14,6.00),vTravel,z5,tPen\WObj:=wPaper;
    MoveL Offs(pOrigin,369.51,107.14,0.00),v60,z0,tPen\WObj:=wPaper;
    MoveL Offs(pOrigin,367.56,109.09,0.00),v40,z0,tPen\WObj:=wPaper;
    MoveL Offs(pOrigin,368.20,108.64,0.00),v40,z0,tPen\WObj:=wPaper;
    MoveL Offs(pOrigin,367.15,107.59,0.00),v40,z0,tPen\WObj:=wPaper;
    MoveL Offs(pOrigin,366.97,106.69,0.00),v40,z0,tPen\WObj:=wPaper;
    MoveL Offs(pOrigin,365.16,108.50,0.00),v40,z0,tPen\WObj:=wPaper;
    MoveL Offs(pOrigin,364.12,108.05,0.00),v40,z0,tPen\WObj:=wPaper;
    MoveL Offs(pOrigin,365.77,106.40,0.00),v40,fine,tPen\WObj:=wPaper;
    MoveL Offs(pOrigin,365.77,106.40,6.00),v60,z5,tPen\WObj:=wPaper;
    MoveL Offs(pOrigin,364.42,106.25,6.00),vTravel,z5,tPen\WObj:=wPaper;
    MoveL Offs(pOrigin,364.42,106.25,0.00),v60,z0,tPen\WObj:=wPaper;
    MoveL Offs(pOrigin,362.92,107.76,0.00),v40,z0,tPen\WObj:=wPaper;
    MoveL Offs(pOrigin,361.87,107.31,0.00),v40,z0,tPen\WObj:=wPaper;
    MoveL Offs(pOrigin,363.37,105.81,0.00),v40,fine,tPen\WObj:=wPaper;
    MoveL Offs(pOrigin,363.37,105.81,6.00),v60,z5,tPen\WObj:=wPaper;
    MoveL Offs(pOrigin,362.18,105.51,6.00),vTravel,z5,tPen\WObj:=wPaper;
    MoveL Offs(pOrigin,362.18,105.51,0.00),v60,z0,tPen\WObj:=wPaper;
    MoveL Offs(pOrigin,360.82,106.86,0.00),v40,z0,tPen\WObj:=wPaper;
    MoveL Offs(pOrigin,359.93,106.27,0.00),v40,z0,tPen\WObj:=wPaper;
    MoveL Offs(pOrigin,360.98,105.21,0.00),v40,z0,tPen\WObj:=wPaper;
    MoveL Offs(pOrigin,359.93,104.77,0.00),v40,z0,tPen\WObj:=wPaper;
    MoveL Offs(pOrigin,358.73,105.97,0.00),v40,fine,tPen\WObj:=wPaper;
    MoveL Offs(pOrigin,358.73,105.97,6.00),v60,z5,tPen\WObj:=wPaper;
    MoveL Offs(pOrigin,357.52,107.93,6.00),vTravel,z5,tPen\WObj:=wPaper;
    MoveL Offs(pOrigin,357.52,107.93,0.00),v60,z0,tPen\WObj:=wPaper;
    MoveL Offs(pOrigin,356.46,107.93,0.00),v40,fine,tPen\WObj:=wPaper;
    MoveL Offs(pOrigin,356.46,107.93,6.00),v60,z5,tPen\WObj:=wPaper;
    MoveL Offs(pOrigin,362.33,102.36,6.00),vTravel,z5,tPen\WObj:=wPaper;
    MoveL Offs(pOrigin,362.33,102.36,0.00),v60,z0,tPen\WObj:=wPaper;
    MoveL Offs(pOrigin,363.99,100.71,0.00),v40,z0,tPen\WObj:=wPaper;
    MoveL Offs(pOrigin,363.83,101.29,0.00),v40,z0,tPen\WObj:=wPaper;
    MoveL Offs(pOrigin,367.14,104.59,0.00),v40,z0,tPen\WObj:=wPaper;
    MoveL Offs(pOrigin,367.27,104.90,0.00),v40,z0,tPen\WObj:=wPaper;
    MoveL Offs(pOrigin,369.37,102.79,0.00),v40,fine,tPen\WObj:=wPaper;
    MoveL Offs(pOrigin,369.37,102.79,6.00),v60,z5,tPen\WObj:=wPaper;
    MoveL Offs(pOrigin,368.31,106.84,6.00),vTravel,z5,tPen\WObj:=wPaper;
    MoveL Offs(pOrigin,368.31,106.84,0.00),v60,z0,tPen\WObj:=wPaper;
    MoveL Offs(pOrigin,366.51,108.64,0.00),v40,fine,tPen\WObj:=wPaper;
    MoveL Offs(pOrigin,366.51,108.64,6.00),v60,z5,tPen\WObj:=wPaper;
    MoveL Offs(pOrigin,368.95,107.89,6.00),vTravel,z5,tPen\WObj:=wPaper;
    MoveL Offs(pOrigin,368.95,107.89,0.00),v60,z0,tPen\WObj:=wPaper;
    MoveL Offs(pOrigin,370.00,108.94,0.00),v40,z0,tPen\WObj:=wPaper;
    MoveL Offs(pOrigin,370.10,109.53,0.00),v40,z0,tPen\WObj:=wPaper;
    MoveL Offs(pOrigin,372.36,107.28,0.00),v40,z0,tPen\WObj:=wPaper;
    MoveL Offs(pOrigin,372.09,108.05,0.00),v40,z0,tPen\WObj:=wPaper;
    MoveL Offs(pOrigin,373.30,109.25,0.00),v40,z0,tPen\WObj:=wPaper;
    MoveL Offs(pOrigin,372.95,109.67,0.00),v40,z0,tPen\WObj:=wPaper;
    MoveL Offs(pOrigin,375.35,107.27,0.00),v40,z0,tPen\WObj:=wPaper;
    MoveL Offs(pOrigin,375.39,108.36,0.00),v40,z0,tPen\WObj:=wPaper;
    MoveL Offs(pOrigin,376.14,109.11,0.00),v40,z0,tPen\WObj:=wPaper;
    MoveL Offs(pOrigin,375.94,109.66,0.00),v40,z0,tPen\WObj:=wPaper;
    MoveL Offs(pOrigin,378.35,107.26,0.00),v40,fine,tPen\WObj:=wPaper;
    MoveL Offs(pOrigin,378.35,107.26,6.00),v60,z5,tPen\WObj:=wPaper;
    MoveL Offs(pOrigin,379.58,108.08,6.00),vTravel,z5,tPen\WObj:=wPaper;
    MoveL Offs(pOrigin,379.58,108.08,0.00),v60,z0,tPen\WObj:=wPaper;
    MoveL Offs(pOrigin,380.33,108.83,0.00),v40,fine,tPen\WObj:=wPaper;
    MoveL Offs(pOrigin,380.33,108.83,6.00),v60,z5,tPen\WObj:=wPaper;
    MoveL Offs(pOrigin,380.00,107.10,6.00),vTravel,z5,tPen\WObj:=wPaper;
    MoveL Offs(pOrigin,380.00,107.10,0.00),v60,z0,tPen\WObj:=wPaper;
    MoveL Offs(pOrigin,377.44,109.66,0.00),v40,fine,tPen\WObj:=wPaper;
    MoveL Offs(pOrigin,377.44,109.66,6.00),v60,z5,tPen\WObj:=wPaper;
    MoveL Offs(pOrigin,373.56,106.08,6.00),vTravel,z5,tPen\WObj:=wPaper;
    MoveL Offs(pOrigin,373.56,106.08,0.00),v60,z0,tPen\WObj:=wPaper;
    MoveL Offs(pOrigin,376.41,103.22,0.00),v40,fine,tPen\WObj:=wPaper;
    MoveL Offs(pOrigin,376.41,103.22,6.00),v60,z5,tPen\WObj:=wPaper;
    MoveL Offs(pOrigin,371.98,108.70,6.00),vTravel,z5,tPen\WObj:=wPaper;
    MoveL Offs(pOrigin,371.98,108.70,0.00),v60,z0,tPen\WObj:=wPaper;
    MoveL Offs(pOrigin,371.55,108.06,0.00),v40,z0,tPen\WObj:=wPaper;
    MoveL Offs(pOrigin,370.91,108.06,0.00),v40,z0,tPen\WObj:=wPaper;
    MoveL Offs(pOrigin,370.70,108.49,0.00),v40,fine,tPen\WObj:=wPaper;
    MoveL Offs(pOrigin,370.70,108.49,6.00),v60,z5,tPen\WObj:=wPaper;
    MoveL Offs(pOrigin,375.77,117.30,6.00),vTravel,z5,tPen\WObj:=wPaper;
    MoveL Offs(pOrigin,375.77,117.30,0.00),v60,z0,tPen\WObj:=wPaper;
    MoveL Offs(pOrigin,374.12,118.96,0.00),v40,z0,tPen\WObj:=wPaper;
    MoveL Offs(pOrigin,375.02,119.55,0.00),v40,z0,tPen\WObj:=wPaper;
    MoveL Offs(pOrigin,376.82,117.75,0.00),v40,z0,tPen\WObj:=wPaper;
    MoveL Offs(pOrigin,376.32,118.25,0.00),v40,z0,tPen\WObj:=wPaper;
    MoveL Offs(pOrigin,378.57,120.51,0.00),v40,z0,tPen\WObj:=wPaper;
    MoveL Offs(pOrigin,379.20,121.34,0.00),v40,z0,tPen\WObj:=wPaper;
    MoveL Offs(pOrigin,380.86,119.68,0.00),v40,z0,tPen\WObj:=wPaper;
    MoveL Offs(pOrigin,381.90,120.13,0.00),v40,z0,tPen\WObj:=wPaper;
    MoveL Offs(pOrigin,380.25,121.78,0.00),v40,fine,tPen\WObj:=wPaper;
    MoveL Offs(pOrigin,380.25,121.78,6.00),v60,z5,tPen\WObj:=wPaper;
    MoveL Offs(pOrigin,381.14,123.88,6.00),vTravel,z5,tPen\WObj:=wPaper;
    MoveL Offs(pOrigin,381.14,123.88,0.00),v60,z0,tPen\WObj:=wPaper;
    MoveL Offs(pOrigin,379.79,125.23,0.00),v40,z0,tPen\WObj:=wPaper;
    MoveL Offs(pOrigin,378.99,124.64,0.00),v40,z0,tPen\WObj:=wPaper;
    MoveL Offs(pOrigin,384.51,125.70,0.00),v40,fine,tPen\WObj:=wPaper;
    MoveL Offs(pOrigin,384.51,125.70,6.00),v60,z5,tPen\WObj:=wPaper;
    MoveL Offs(pOrigin,385.94,123.56,6.00),vTravel,z5,tPen\WObj:=wPaper;
    MoveL Offs(pOrigin,385.94,123.56,0.00),v60,z0,tPen\WObj:=wPaper;
    MoveL Offs(pOrigin,386.84,122.66,0.00),v40,fine,tPen\WObj:=wPaper;
  ENDPROC

  PROC DrawPart213()
    MoveL Offs(pOrigin,386.84,122.66,6.00),v60,z5,tPen\WObj:=wPaper;
    MoveL Offs(pOrigin,383.85,121.17,6.00),vTravel,z5,tPen\WObj:=wPaper;
    MoveL Offs(pOrigin,383.85,121.17,0.00),v60,z0,tPen\WObj:=wPaper;
    MoveL Offs(pOrigin,382.35,122.68,0.00),v40,fine,tPen\WObj:=wPaper;
    MoveL Offs(pOrigin,382.35,122.68,6.00),v60,z5,tPen\WObj:=wPaper;
    MoveL Offs(pOrigin,382.34,124.17,6.00),vTravel,z5,tPen\WObj:=wPaper;
    MoveL Offs(pOrigin,382.34,124.17,0.00),v60,z0,tPen\WObj:=wPaper;
    MoveL Offs(pOrigin,380.84,125.68,0.00),v40,fine,tPen\WObj:=wPaper;
    MoveL Offs(pOrigin,380.84,125.68,6.00),v60,z5,tPen\WObj:=wPaper;
    MoveL Offs(pOrigin,387.72,127.75,6.00),vTravel,z5,tPen\WObj:=wPaper;
    MoveL Offs(pOrigin,387.72,127.75,0.00),v60,z0,tPen\WObj:=wPaper;
    MoveL Offs(pOrigin,389.83,125.65,0.00),v40,fine,tPen\WObj:=wPaper;
    MoveL Offs(pOrigin,389.83,125.65,6.00),v60,z5,tPen\WObj:=wPaper;
    MoveL Offs(pOrigin,391.17,125.79,6.00),vTravel,z5,tPen\WObj:=wPaper;
    MoveL Offs(pOrigin,391.17,125.79,0.00),v60,z0,tPen\WObj:=wPaper;
    MoveL Offs(pOrigin,388.62,128.35,0.00),v40,fine,tPen\WObj:=wPaper;
    MoveL Offs(pOrigin,388.62,128.35,6.00),v60,z5,tPen\WObj:=wPaper;
    MoveL Offs(pOrigin,389.61,130.10,6.00),vTravel,z5,tPen\WObj:=wPaper;
    MoveL Offs(pOrigin,389.61,130.10,0.00),v60,z0,tPen\WObj:=wPaper;
    MoveL Offs(pOrigin,391.10,130.10,0.00),v40,fine,tPen\WObj:=wPaper;
    MoveL Offs(pOrigin,391.10,130.10,6.00),v60,z5,tPen\WObj:=wPaper;
    MoveL Offs(pOrigin,392.85,128.89,6.00),vTravel,z5,tPen\WObj:=wPaper;
    MoveL Offs(pOrigin,392.85,128.89,0.00),v60,z0,tPen\WObj:=wPaper;
    MoveL Offs(pOrigin,392.85,127.61,0.00),v40,fine,tPen\WObj:=wPaper;
    MoveL Offs(pOrigin,392.85,127.61,6.00),v60,z5,tPen\WObj:=wPaper;
    MoveL Offs(pOrigin,394.71,126.34,6.00),vTravel,z5,tPen\WObj:=wPaper;
    MoveL Offs(pOrigin,394.71,126.34,0.00),v60,z0,tPen\WObj:=wPaper;
    MoveL Offs(pOrigin,394.50,126.76,0.00),v40,z0,tPen\WObj:=wPaper;
    MoveL Offs(pOrigin,394.71,126.34,0.00),v40,z0,tPen\WObj:=wPaper;
    MoveL Offs(pOrigin,395.14,125.88,0.00),v40,z0,tPen\WObj:=wPaper;
    MoveL Offs(pOrigin,396.41,125.88,0.00),v40,z0,tPen\WObj:=wPaper;
    MoveL Offs(pOrigin,396.62,124.82,0.00),v40,z0,tPen\WObj:=wPaper;
    MoveL Offs(pOrigin,395.56,124.82,0.00),v40,z0,tPen\WObj:=wPaper;
    MoveL Offs(pOrigin,395.56,123.77,0.00),v40,z0,tPen\WObj:=wPaper;
    MoveL Offs(pOrigin,396.62,123.77,0.00),v40,z0,tPen\WObj:=wPaper;
    MoveL Offs(pOrigin,396.62,122.71,0.00),v40,z0,tPen\WObj:=wPaper;
    MoveL Offs(pOrigin,395.56,122.71,0.00),v40,fine,tPen\WObj:=wPaper;
    MoveL Offs(pOrigin,395.56,122.71,6.00),v60,z5,tPen\WObj:=wPaper;
    MoveL Offs(pOrigin,397.63,122.33,6.00),vTravel,z5,tPen\WObj:=wPaper;
    MoveL Offs(pOrigin,397.63,122.33,0.00),v60,z0,tPen\WObj:=wPaper;
    MoveL Offs(pOrigin,388.46,131.50,0.00),v40,fine,tPen\WObj:=wPaper;
    MoveL Offs(pOrigin,388.46,131.50,6.00),v60,z5,tPen\WObj:=wPaper;
    MoveL Offs(pOrigin,392.16,135.38,6.00),vTravel,z5,tPen\WObj:=wPaper;
    MoveL Offs(pOrigin,392.16,135.38,0.00),v60,z0,tPen\WObj:=wPaper;
    MoveL Offs(pOrigin,393.44,135.38,0.00),v40,z0,tPen\WObj:=wPaper;
    MoveL Offs(pOrigin,393.22,136.44,0.00),v40,z0,tPen\WObj:=wPaper;
    MoveL Offs(pOrigin,392.16,136.44,0.00),v40,fine,tPen\WObj:=wPaper;
    MoveL Offs(pOrigin,392.16,136.44,6.00),v60,z5,tPen\WObj:=wPaper;
    MoveL Offs(pOrigin,393.82,141.07,6.00),vTravel,z5,tPen\WObj:=wPaper;
    MoveL Offs(pOrigin,393.82,141.07,0.00),v60,z0,tPen\WObj:=wPaper;
    MoveL Offs(pOrigin,390.07,144.82,0.00),v40,fine,tPen\WObj:=wPaper;
    MoveL Offs(pOrigin,390.07,144.82,6.00),v60,z5,tPen\WObj:=wPaper;
    MoveL Offs(pOrigin,389.91,147.97,6.00),vTravel,z5,tPen\WObj:=wPaper;
    MoveL Offs(pOrigin,389.91,147.97,0.00),v60,z0,tPen\WObj:=wPaper;
    MoveL Offs(pOrigin,393.36,144.51,0.00),v40,fine,tPen\WObj:=wPaper;
    MoveL Offs(pOrigin,393.36,144.51,6.00),v60,z5,tPen\WObj:=wPaper;
    MoveL Offs(pOrigin,391.74,151.22,6.00),vTravel,z5,tPen\WObj:=wPaper;
    MoveL Offs(pOrigin,391.74,151.22,0.00),v60,z0,tPen\WObj:=wPaper;
    MoveL Offs(pOrigin,390.67,151.22,0.00),v40,fine,tPen\WObj:=wPaper;
    MoveL Offs(pOrigin,390.67,151.22,6.00),v60,z5,tPen\WObj:=wPaper;
    MoveL Offs(pOrigin,392.13,156.20,6.00),vTravel,z5,tPen\WObj:=wPaper;
    MoveL Offs(pOrigin,392.13,156.20,0.00),v60,z0,tPen\WObj:=wPaper;
    MoveL Offs(pOrigin,388.67,159.66,0.00),v40,fine,tPen\WObj:=wPaper;
    MoveL Offs(pOrigin,388.67,159.66,6.00),v60,z5,tPen\WObj:=wPaper;
    MoveL Offs(pOrigin,389.83,160.73,6.00),vTravel,z5,tPen\WObj:=wPaper;
    MoveL Offs(pOrigin,389.83,160.73,0.00),v60,z0,tPen\WObj:=wPaper;
    MoveL Offs(pOrigin,390.89,160.73,0.00),v40,fine,tPen\WObj:=wPaper;
    MoveL Offs(pOrigin,390.89,160.73,6.00),v60,z5,tPen\WObj:=wPaper;
    MoveL Offs(pOrigin,391.66,162.64,6.00),vTravel,z5,tPen\WObj:=wPaper;
    MoveL Offs(pOrigin,391.66,162.64,0.00),v60,z0,tPen\WObj:=wPaper;
    MoveL Offs(pOrigin,388.20,166.10,0.00),v40,fine,tPen\WObj:=wPaper;
    MoveL Offs(pOrigin,388.20,166.10,6.00),v60,z5,tPen\WObj:=wPaper;
    MoveL Offs(pOrigin,389.40,164.95,6.00),vTravel,z5,tPen\WObj:=wPaper;
    MoveL Offs(pOrigin,389.40,164.95,0.00),v60,z0,tPen\WObj:=wPaper;
    MoveL Offs(pOrigin,390.46,164.95,0.00),v40,fine,tPen\WObj:=wPaper;
    MoveL Offs(pOrigin,390.46,164.95,6.00),v60,z5,tPen\WObj:=wPaper;
    MoveL Offs(pOrigin,390.89,169.39,6.00),vTravel,z5,tPen\WObj:=wPaper;
    MoveL Offs(pOrigin,390.89,169.39,0.00),v60,z0,tPen\WObj:=wPaper;
    MoveL Offs(pOrigin,387.58,172.69,0.00),v40,fine,tPen\WObj:=wPaper;
    MoveL Offs(pOrigin,387.58,172.69,6.00),v60,z5,tPen\WObj:=wPaper;
    MoveL Offs(pOrigin,388.76,171.29,6.00),vTravel,z5,tPen\WObj:=wPaper;
    MoveL Offs(pOrigin,388.76,171.29,0.00),v60,z0,tPen\WObj:=wPaper;
    MoveL Offs(pOrigin,389.83,171.29,0.00),v40,fine,tPen\WObj:=wPaper;
    MoveL Offs(pOrigin,389.83,171.29,6.00),v60,z5,tPen\WObj:=wPaper;
    MoveL Offs(pOrigin,390.43,174.33,6.00),vTravel,z5,tPen\WObj:=wPaper;
    MoveL Offs(pOrigin,390.43,174.33,0.00),v60,z0,tPen\WObj:=wPaper;
    MoveL Offs(pOrigin,387.12,177.64,0.00),v40,fine,tPen\WObj:=wPaper;
    MoveL Offs(pOrigin,387.12,177.64,6.00),v60,z5,tPen\WObj:=wPaper;
    MoveL Offs(pOrigin,387.59,178.81,6.00),vTravel,z5,tPen\WObj:=wPaper;
    MoveL Offs(pOrigin,387.59,178.81,0.00),v60,z0,tPen\WObj:=wPaper;
    MoveL Offs(pOrigin,389.39,180.61,0.00),v40,z0,tPen\WObj:=wPaper;
    MoveL Offs(pOrigin,389.81,180.92,0.00),v40,z0,tPen\WObj:=wPaper;
    MoveL Offs(pOrigin,386.50,184.23,0.00),v40,z0,tPen\WObj:=wPaper;
    MoveL Offs(pOrigin,387.16,184.35,0.00),v40,z0,tPen\WObj:=wPaper;
    MoveL Offs(pOrigin,388.81,186.00,0.00),v40,fine,tPen\WObj:=wPaper;
    MoveL Offs(pOrigin,388.81,186.00,6.00),v60,z5,tPen\WObj:=wPaper;
    MoveL Offs(pOrigin,388.34,187.13,6.00),vTravel,z5,tPen\WObj:=wPaper;
    MoveL Offs(pOrigin,388.34,187.13,0.00),v60,z0,tPen\WObj:=wPaper;
    MoveL Offs(pOrigin,387.28,187.13,0.00),v40,z0,tPen\WObj:=wPaper;
    MoveL Offs(pOrigin,386.87,187.04,0.00),v40,z0,tPen\WObj:=wPaper;
    MoveL Offs(pOrigin,388.52,188.69,0.00),v40,z0,tPen\WObj:=wPaper;
    MoveL Offs(pOrigin,388.12,189.24,0.00),v40,z0,tPen\WObj:=wPaper;
    MoveL Offs(pOrigin,387.06,189.24,0.00),v40,fine,tPen\WObj:=wPaper;
    MoveL Offs(pOrigin,387.06,189.24,6.00),v60,z5,tPen\WObj:=wPaper;
    MoveL Offs(pOrigin,389.18,189.02,6.00),vTravel,z5,tPen\WObj:=wPaper;
    MoveL Offs(pOrigin,389.18,189.02,0.00),v60,z0,tPen\WObj:=wPaper;
    MoveL Offs(pOrigin,385.58,192.62,0.00),v40,fine,tPen\WObj:=wPaper;
    MoveL Offs(pOrigin,385.58,192.62,6.00),v60,z5,tPen\WObj:=wPaper;
    MoveL Offs(pOrigin,385.85,196.48,6.00),vTravel,z5,tPen\WObj:=wPaper;
    MoveL Offs(pOrigin,385.85,196.48,0.00),v60,z0,tPen\WObj:=wPaper;
    MoveL Offs(pOrigin,387.65,198.28,0.00),v40,fine,tPen\WObj:=wPaper;
    MoveL Offs(pOrigin,387.65,198.28,6.00),v60,z5,tPen\WObj:=wPaper;
    MoveL Offs(pOrigin,381.51,198.18,6.00),vTravel,z5,tPen\WObj:=wPaper;
    MoveL Offs(pOrigin,381.51,198.18,0.00),v60,z0,tPen\WObj:=wPaper;
    MoveL Offs(pOrigin,379.11,200.58,0.00),v40,z0,tPen\WObj:=wPaper;
    MoveL Offs(pOrigin,379.42,200.50,0.00),v40,z0,tPen\WObj:=wPaper;
    MoveL Offs(pOrigin,381.52,202.60,0.00),v40,z0,tPen\WObj:=wPaper;
    MoveL Offs(pOrigin,381.80,202.37,0.00),v40,z0,tPen\WObj:=wPaper;
    MoveL Offs(pOrigin,379.25,204.93,0.00),v40,z0,tPen\WObj:=wPaper;
    MoveL Offs(pOrigin,379.88,205.45,0.00),v40,z0,tPen\WObj:=wPaper;
  ENDPROC

  PROC DrawPart214()
    MoveL Offs(pOrigin,381.68,207.25,0.00),v40,fine,tPen\WObj:=wPaper;
    MoveL Offs(pOrigin,381.68,207.25,6.00),v60,z5,tPen\WObj:=wPaper;
    MoveL Offs(pOrigin,379.39,206.27,6.00),vTravel,z5,tPen\WObj:=wPaper;
    MoveL Offs(pOrigin,379.39,206.27,0.00),v60,z0,tPen\WObj:=wPaper;
    MoveL Offs(pOrigin,382.10,203.57,0.00),v40,z0,tPen\WObj:=wPaper;
    MoveL Offs(pOrigin,381.53,204.10,0.00),v40,z0,tPen\WObj:=wPaper;
    MoveL Offs(pOrigin,379.72,202.30,0.00),v40,fine,tPen\WObj:=wPaper;
    MoveL Offs(pOrigin,379.72,202.30,6.00),v60,z5,tPen\WObj:=wPaper;
    MoveL Offs(pOrigin,376.57,200.14,6.00),vTravel,z5,tPen\WObj:=wPaper;
    MoveL Offs(pOrigin,376.57,200.14,0.00),v60,z0,tPen\WObj:=wPaper;
    MoveL Offs(pOrigin,374.16,202.54,0.00),v40,fine,tPen\WObj:=wPaper;
    MoveL Offs(pOrigin,374.16,202.54,6.00),v60,z5,tPen\WObj:=wPaper;
    MoveL Offs(pOrigin,373.57,200.15,6.00),vTravel,z5,tPen\WObj:=wPaper;
    MoveL Offs(pOrigin,373.57,200.15,0.00),v60,z0,tPen\WObj:=wPaper;
    MoveL Offs(pOrigin,376.12,197.59,0.00),v40,fine,tPen\WObj:=wPaper;
    MoveL Offs(pOrigin,376.12,197.59,6.00),v60,z5,tPen\WObj:=wPaper;
    MoveL Offs(pOrigin,373.72,197.79,6.00),vTravel,z5,tPen\WObj:=wPaper;
    MoveL Offs(pOrigin,373.72,197.79,0.00),v60,z0,tPen\WObj:=wPaper;
    MoveL Offs(pOrigin,375.97,200.04,0.00),v40,fine,tPen\WObj:=wPaper;
    MoveL Offs(pOrigin,375.97,200.04,6.00),v60,z5,tPen\WObj:=wPaper;
    MoveL Offs(pOrigin,373.13,197.60,6.00),vTravel,z5,tPen\WObj:=wPaper;
    MoveL Offs(pOrigin,373.13,197.60,0.00),v60,z0,tPen\WObj:=wPaper;
    MoveL Offs(pOrigin,375.53,195.20,0.00),v40,fine,tPen\WObj:=wPaper;
    MoveL Offs(pOrigin,375.53,195.20,6.00),v60,z5,tPen\WObj:=wPaper;
    MoveL Offs(pOrigin,378.67,196.54,6.00),vTravel,z5,tPen\WObj:=wPaper;
    MoveL Offs(pOrigin,378.67,196.54,0.00),v60,z0,tPen\WObj:=wPaper;
    MoveL Offs(pOrigin,381.08,194.13,0.00),v40,fine,tPen\WObj:=wPaper;
    MoveL Offs(pOrigin,381.08,194.13,6.00),v60,z5,tPen\WObj:=wPaper;
    MoveL Offs(pOrigin,377.80,189.95,6.00),vTravel,z5,tPen\WObj:=wPaper;
    MoveL Offs(pOrigin,377.80,189.95,0.00),v60,z0,tPen\WObj:=wPaper;
    MoveL Offs(pOrigin,379.90,187.85,0.00),v40,fine,tPen\WObj:=wPaper;
    MoveL Offs(pOrigin,379.90,187.85,6.00),v60,z5,tPen\WObj:=wPaper;
    MoveL Offs(pOrigin,374.89,190.00,6.00),vTravel,z5,tPen\WObj:=wPaper;
    MoveL Offs(pOrigin,374.89,190.00,0.00),v60,z0,tPen\WObj:=wPaper;
    MoveL Offs(pOrigin,373.39,188.50,0.00),v40,fine,tPen\WObj:=wPaper;
    MoveL Offs(pOrigin,373.39,188.50,6.00),v60,z5,tPen\WObj:=wPaper;
    MoveL Offs(pOrigin,374.64,191.61,6.00),vTravel,z5,tPen\WObj:=wPaper;
    MoveL Offs(pOrigin,374.64,191.61,0.00),v60,z0,tPen\WObj:=wPaper;
    MoveL Offs(pOrigin,372.24,194.01,0.00),v40,fine,tPen\WObj:=wPaper;
    MoveL Offs(pOrigin,372.24,194.01,6.00),v60,z5,tPen\WObj:=wPaper;
    MoveL Offs(pOrigin,377.89,207.78,6.00),vTravel,z5,tPen\WObj:=wPaper;
    MoveL Offs(pOrigin,377.89,207.78,0.00),v60,z0,tPen\WObj:=wPaper;
    MoveL Offs(pOrigin,375.04,210.63,0.00),v40,z0,tPen\WObj:=wPaper;
    MoveL Offs(pOrigin,375.55,210.08,0.00),v40,z0,tPen\WObj:=wPaper;
    MoveL Offs(pOrigin,377.66,212.18,0.00),v40,z0,tPen\WObj:=wPaper;
    MoveL Offs(pOrigin,377.29,212.47,0.00),v40,z0,tPen\WObj:=wPaper;
    MoveL Offs(pOrigin,376.22,212.47,0.00),v40,fine,tPen\WObj:=wPaper;
    MoveL Offs(pOrigin,376.22,212.47,6.00),v60,z5,tPen\WObj:=wPaper;
    MoveL Offs(pOrigin,374.73,212.43,6.00),vTravel,z5,tPen\WObj:=wPaper;
    MoveL Offs(pOrigin,374.73,212.43,0.00),v60,z0,tPen\WObj:=wPaper;
    MoveL Offs(pOrigin,377.89,209.27,0.00),v40,fine,tPen\WObj:=wPaper;
    MoveL Offs(pOrigin,377.89,209.27,6.00),v60,z5,tPen\WObj:=wPaper;
    MoveL Offs(pOrigin,377.08,210.36,6.00),vTravel,z5,tPen\WObj:=wPaper;
    MoveL Offs(pOrigin,377.08,210.36,0.00),v60,z0,tPen\WObj:=wPaper;
    MoveL Offs(pOrigin,376.01,210.36,0.00),v40,fine,tPen\WObj:=wPaper;
    MoveL Offs(pOrigin,376.01,210.36,6.00),v60,z5,tPen\WObj:=wPaper;
    MoveL Offs(pOrigin,378.03,210.62,6.00),vTravel,z5,tPen\WObj:=wPaper;
    MoveL Offs(pOrigin,378.03,210.62,0.00),v60,z0,tPen\WObj:=wPaper;
    MoveL Offs(pOrigin,374.73,213.93,0.00),v40,fine,tPen\WObj:=wPaper;
    MoveL Offs(pOrigin,374.73,213.93,6.00),v60,z5,tPen\WObj:=wPaper;
    MoveL Offs(pOrigin,374.57,215.58,6.00),vTravel,z5,tPen\WObj:=wPaper;
    MoveL Offs(pOrigin,374.57,215.58,0.00),v60,z0,tPen\WObj:=wPaper;
    MoveL Offs(pOrigin,378.18,211.97,0.00),v40,fine,tPen\WObj:=wPaper;
    MoveL Offs(pOrigin,378.18,211.97,6.00),v60,z5,tPen\WObj:=wPaper;
    MoveL Offs(pOrigin,380.21,216.23,6.00),vTravel,z5,tPen\WObj:=wPaper;
    MoveL Offs(pOrigin,380.21,216.23,0.00),v60,z0,tPen\WObj:=wPaper;
    MoveL Offs(pOrigin,381.72,217.74,0.00),v40,fine,tPen\WObj:=wPaper;
    MoveL Offs(pOrigin,381.72,217.74,6.00),v60,z5,tPen\WObj:=wPaper;
    MoveL Offs(pOrigin,383.37,220.89,6.00),vTravel,z5,tPen\WObj:=wPaper;
    MoveL Offs(pOrigin,383.37,220.89,0.00),v60,z0,tPen\WObj:=wPaper;
    MoveL Offs(pOrigin,385.18,222.69,0.00),v40,z0,tPen\WObj:=wPaper;
    MoveL Offs(pOrigin,384.73,223.74,0.00),v40,z0,tPen\WObj:=wPaper;
    MoveL Offs(pOrigin,383.23,222.23,0.00),v40,fine,tPen\WObj:=wPaper;
    MoveL Offs(pOrigin,383.23,222.23,6.00),v60,z5,tPen\WObj:=wPaper;
    MoveL Offs(pOrigin,382.34,225.83,6.00),vTravel,z5,tPen\WObj:=wPaper;
    MoveL Offs(pOrigin,382.34,225.83,0.00),v60,z0,tPen\WObj:=wPaper;
    MoveL Offs(pOrigin,383.84,227.33,0.00),v40,z0,tPen\WObj:=wPaper;
    MoveL Offs(pOrigin,383.66,227.27,0.00),v40,z0,tPen\WObj:=wPaper;
    MoveL Offs(pOrigin,383.45,227.70,0.00),v40,z0,tPen\WObj:=wPaper;
    MoveL Offs(pOrigin,383.66,227.27,0.00),v40,fine,tPen\WObj:=wPaper;
    MoveL Offs(pOrigin,383.66,227.27,6.00),v60,z5,tPen\WObj:=wPaper;
    MoveL Offs(pOrigin,382.95,229.42,6.00),vTravel,z5,tPen\WObj:=wPaper;
    MoveL Offs(pOrigin,382.95,229.42,0.00),v60,z0,tPen\WObj:=wPaper;
    MoveL Offs(pOrigin,379.35,225.82,0.00),v40,fine,tPen\WObj:=wPaper;
    MoveL Offs(pOrigin,379.35,225.82,6.00),v60,z5,tPen\WObj:=wPaper;
    MoveL Offs(pOrigin,376.21,230.15,6.00),vTravel,z5,tPen\WObj:=wPaper;
    MoveL Offs(pOrigin,376.21,230.15,0.00),v60,z0,tPen\WObj:=wPaper;
    MoveL Offs(pOrigin,374.86,228.80,0.00),v40,fine,tPen\WObj:=wPaper;
    MoveL Offs(pOrigin,374.86,228.80,6.00),v60,z5,tPen\WObj:=wPaper;
    MoveL Offs(pOrigin,374.10,230.68,6.00),vTravel,z5,tPen\WObj:=wPaper;
    MoveL Offs(pOrigin,374.10,230.68,0.00),v60,z0,tPen\WObj:=wPaper;
    MoveL Offs(pOrigin,373.89,231.10,0.00),v40,z0,tPen\WObj:=wPaper;
    MoveL Offs(pOrigin,374.10,230.68,0.00),v40,fine,tPen\WObj:=wPaper;
    MoveL Offs(pOrigin,374.10,230.68,6.00),v60,z5,tPen\WObj:=wPaper;
    MoveL Offs(pOrigin,370.49,229.40,6.00),vTravel,z5,tPen\WObj:=wPaper;
    MoveL Offs(pOrigin,370.49,229.40,0.00),v60,z0,tPen\WObj:=wPaper;
    MoveL Offs(pOrigin,369.85,230.04,0.00),v40,z0,tPen\WObj:=wPaper;
    MoveL Offs(pOrigin,370.49,229.40,0.00),v40,fine,tPen\WObj:=wPaper;
    MoveL Offs(pOrigin,370.49,229.40,6.00),v60,z5,tPen\WObj:=wPaper;
    MoveL Offs(pOrigin,369.64,230.25,6.00),vTravel,z5,tPen\WObj:=wPaper;
    MoveL Offs(pOrigin,369.64,230.25,0.00),v60,z0,tPen\WObj:=wPaper;
    MoveL Offs(pOrigin,369.00,230.89,0.00),v40,z0,tPen\WObj:=wPaper;
    MoveL Offs(pOrigin,369.64,230.25,0.00),v40,fine,tPen\WObj:=wPaper;
    MoveL Offs(pOrigin,369.64,230.25,6.00),v60,z5,tPen\WObj:=wPaper;
    MoveL Offs(pOrigin,359.02,241.33,6.00),vTravel,z5,tPen\WObj:=wPaper;
    MoveL Offs(pOrigin,359.02,241.33,0.00),v60,z0,tPen\WObj:=wPaper;
    MoveL Offs(pOrigin,360.82,243.14,0.00),v40,fine,tPen\WObj:=wPaper;
    MoveL Offs(pOrigin,360.82,243.14,6.00),v60,z5,tPen\WObj:=wPaper;
    MoveL Offs(pOrigin,386.06,216.10,6.00),vTravel,z5,tPen\WObj:=wPaper;
    MoveL Offs(pOrigin,386.06,216.10,0.00),v60,z0,tPen\WObj:=wPaper;
    MoveL Offs(pOrigin,384.40,214.45,0.00),v40,fine,tPen\WObj:=wPaper;
    MoveL Offs(pOrigin,384.40,214.45,6.00),v60,z5,tPen\WObj:=wPaper;
    MoveL Offs(pOrigin,339.18,179.28,6.00),vTravel,z5,tPen\WObj:=wPaper;
    MoveL Offs(pOrigin,339.18,179.28,0.00),v60,z0,tPen\WObj:=wPaper;
    MoveL Offs(pOrigin,338.43,180.03,0.00),v40,z0,tPen\WObj:=wPaper;
    MoveL Offs(pOrigin,337.53,179.44,0.00),v40,z0,tPen\WObj:=wPaper;
    MoveL Offs(pOrigin,338.43,178.54,0.00),v40,z0,tPen\WObj:=wPaper;
    MoveL Offs(pOrigin,337.54,177.94,0.00),v40,z0,tPen\WObj:=wPaper;
    MoveL Offs(pOrigin,336.63,178.84,0.00),v40,z0,tPen\WObj:=wPaper;
    MoveL Offs(pOrigin,335.89,178.09,0.00),v40,z0,tPen\WObj:=wPaper;
  ENDPROC

  PROC DrawPart215()
    MoveL Offs(pOrigin,336.94,177.04,0.00),v40,z0,tPen\WObj:=wPaper;
    MoveL Offs(pOrigin,336.04,176.45,0.00),v40,z0,tPen\WObj:=wPaper;
    MoveL Offs(pOrigin,334.99,177.50,0.00),v40,z0,tPen\WObj:=wPaper;
    MoveL Offs(pOrigin,334.09,176.90,0.00),v40,z0,tPen\WObj:=wPaper;
    MoveL Offs(pOrigin,335.45,175.55,0.00),v40,z0,tPen\WObj:=wPaper;
    MoveL Offs(pOrigin,334.55,174.95,0.00),v40,z0,tPen\WObj:=wPaper;
    MoveL Offs(pOrigin,333.50,176.00,0.00),v40,z0,tPen\WObj:=wPaper;
    MoveL Offs(pOrigin,332.60,175.41,0.00),v40,z0,tPen\WObj:=wPaper;
    MoveL Offs(pOrigin,333.95,174.06,0.00),v40,z0,tPen\WObj:=wPaper;
    MoveL Offs(pOrigin,333.06,173.46,0.00),v40,z0,tPen\WObj:=wPaper;
    MoveL Offs(pOrigin,331.70,174.81,0.00),v40,z0,tPen\WObj:=wPaper;
    MoveL Offs(pOrigin,331.11,173.91,0.00),v40,z0,tPen\WObj:=wPaper;
    MoveL Offs(pOrigin,332.46,172.56,0.00),v40,z0,tPen\WObj:=wPaper;
    MoveL Offs(pOrigin,331.56,171.97,0.00),v40,z0,tPen\WObj:=wPaper;
    MoveL Offs(pOrigin,330.21,173.32,0.00),v40,z0,tPen\WObj:=wPaper;
    MoveL Offs(pOrigin,329.61,172.42,0.00),v40,z0,tPen\WObj:=wPaper;
    MoveL Offs(pOrigin,330.97,171.07,0.00),v40,z0,tPen\WObj:=wPaper;
    MoveL Offs(pOrigin,330.22,170.32,0.00),v40,z0,tPen\WObj:=wPaper;
    MoveL Offs(pOrigin,328.72,171.82,0.00),v40,z0,tPen\WObj:=wPaper;
    MoveL Offs(pOrigin,329.75,171.74,0.00),v40,z0,tPen\WObj:=wPaper;
    MoveL Offs(pOrigin,327.94,169.93,0.00),v40,z0,tPen\WObj:=wPaper;
    MoveL Offs(pOrigin,327.37,170.18,0.00),v40,z0,tPen\WObj:=wPaper;
    MoveL Offs(pOrigin,328.88,168.68,0.00),v40,z0,tPen\WObj:=wPaper;
    MoveL Offs(pOrigin,329.62,169.43,0.00),v40,z0,tPen\WObj:=wPaper;
    MoveL Offs(pOrigin,328.12,170.93,0.00),v40,fine,tPen\WObj:=wPaper;
    MoveL Offs(pOrigin,328.12,170.93,6.00),v60,z5,tPen\WObj:=wPaper;
    MoveL Offs(pOrigin,326.63,169.43,6.00),vTravel,z5,tPen\WObj:=wPaper;
    MoveL Offs(pOrigin,326.63,169.43,0.00),v60,z0,tPen\WObj:=wPaper;
    MoveL Offs(pOrigin,328.28,167.78,0.00),v40,fine,tPen\WObj:=wPaper;
    MoveL Offs(pOrigin,328.28,167.78,6.00),v60,z5,tPen\WObj:=wPaper;
    MoveL Offs(pOrigin,331.17,172.66,6.00),vTravel,z5,tPen\WObj:=wPaper;
    MoveL Offs(pOrigin,331.17,172.66,0.00),v60,z0,tPen\WObj:=wPaper;
    MoveL Offs(pOrigin,332.02,173.51,0.00),v40,z0,tPen\WObj:=wPaper;
    MoveL Offs(pOrigin,331.17,172.66,0.00),v40,fine,tPen\WObj:=wPaper;
    MoveL Offs(pOrigin,331.17,172.66,6.00),v60,z5,tPen\WObj:=wPaper;
    MoveL Offs(pOrigin,332.66,174.15,6.00),vTravel,z5,tPen\WObj:=wPaper;
    MoveL Offs(pOrigin,332.66,174.15,0.00),v60,z0,tPen\WObj:=wPaper;
    MoveL Offs(pOrigin,333.51,175.00,0.00),v40,z0,tPen\WObj:=wPaper;
    MoveL Offs(pOrigin,332.66,174.15,0.00),v40,fine,tPen\WObj:=wPaper;
    MoveL Offs(pOrigin,332.66,174.15,6.00),v60,z5,tPen\WObj:=wPaper;
    MoveL Offs(pOrigin,321.80,181.73,6.00),vTravel,z5,tPen\WObj:=wPaper;
    MoveL Offs(pOrigin,321.80,181.73,0.00),v60,z0,tPen\WObj:=wPaper;
    MoveL Offs(pOrigin,319.39,184.14,0.00),v40,fine,tPen\WObj:=wPaper;
    MoveL Offs(pOrigin,319.39,184.14,6.00),v60,z5,tPen\WObj:=wPaper;
    MoveL Offs(pOrigin,320.55,184.56,6.00),vTravel,z5,tPen\WObj:=wPaper;
    MoveL Offs(pOrigin,320.55,184.56,0.00),v60,z0,tPen\WObj:=wPaper;
    MoveL Offs(pOrigin,320.12,184.99,0.00),v40,z0,tPen\WObj:=wPaper;
    MoveL Offs(pOrigin,320.34,185.84,0.00),v40,z0,tPen\WObj:=wPaper;
    MoveL Offs(pOrigin,319.90,185.79,0.00),v40,z0,tPen\WObj:=wPaper;
    MoveL Offs(pOrigin,320.65,186.54,0.00),v40,z0,tPen\WObj:=wPaper;
    MoveL Offs(pOrigin,321.33,186.68,0.00),v40,z0,tPen\WObj:=wPaper;
    MoveL Offs(pOrigin,318.18,189.83,0.00),v40,fine,tPen\WObj:=wPaper;
    MoveL Offs(pOrigin,318.18,189.83,6.00),v60,z5,tPen\WObj:=wPaper;
    MoveL Offs(pOrigin,318.93,187.58,6.00),vTravel,z5,tPen\WObj:=wPaper;
    MoveL Offs(pOrigin,318.93,187.58,0.00),v60,z0,tPen\WObj:=wPaper;
    MoveL Offs(pOrigin,321.64,184.88,0.00),v40,fine,tPen\WObj:=wPaper;
    MoveL Offs(pOrigin,321.64,184.88,6.00),v60,z5,tPen\WObj:=wPaper;
    MoveL Offs(pOrigin,320.94,183.84,6.00),vTravel,z5,tPen\WObj:=wPaper;
    MoveL Offs(pOrigin,320.94,183.84,0.00),v60,z0,tPen\WObj:=wPaper;
    MoveL Offs(pOrigin,320.19,183.09,0.00),v40,z0,tPen\WObj:=wPaper;
    MoveL Offs(pOrigin,320.55,183.50,0.00),v40,z0,tPen\WObj:=wPaper;
    MoveL Offs(pOrigin,321.19,182.86,0.00),v40,z0,tPen\WObj:=wPaper;
    MoveL Offs(pOrigin,320.55,181.59,0.00),v40,z0,tPen\WObj:=wPaper;
    MoveL Offs(pOrigin,320.55,179.25,0.00),v40,z0,tPen\WObj:=wPaper;
    MoveL Offs(pOrigin,318.00,170.32,0.00),v40,fine,tPen\WObj:=wPaper;
    MoveL Offs(pOrigin,318.00,170.32,6.00),v60,z5,tPen\WObj:=wPaper;
    MoveL Offs(pOrigin,306.70,169.94,6.00),vTravel,z5,tPen\WObj:=wPaper;
    MoveL Offs(pOrigin,306.70,169.94,0.00),v60,z0,tPen\WObj:=wPaper;
    MoveL Offs(pOrigin,305.50,171.15,0.00),v40,z0,tPen\WObj:=wPaper;
    MoveL Offs(pOrigin,304.88,170.76,0.00),v40,z0,tPen\WObj:=wPaper;
    MoveL Offs(pOrigin,303.52,169.41,0.00),v40,z0,tPen\WObj:=wPaper;
    MoveL Offs(pOrigin,303.86,168.31,0.00),v40,z0,tPen\WObj:=wPaper;
    MoveL Offs(pOrigin,298.45,173.72,0.00),v40,z0,tPen\WObj:=wPaper;
    MoveL Offs(pOrigin,298.29,173.14,0.00),v40,z0,tPen\WObj:=wPaper;
    MoveL Offs(pOrigin,297.09,171.94,0.00),v40,z0,tPen\WObj:=wPaper;
    MoveL Offs(pOrigin,296.21,171.48,0.00),v40,z0,tPen\WObj:=wPaper;
    MoveL Offs(pOrigin,294.71,172.98,0.00),v40,z0,tPen\WObj:=wPaper;
    MoveL Offs(pOrigin,295.15,174.02,0.00),v40,z0,tPen\WObj:=wPaper;
    MoveL Offs(pOrigin,299.21,169.97,0.00),v40,z0,tPen\WObj:=wPaper;
    MoveL Offs(pOrigin,299.18,171.04,0.00),v40,z0,tPen\WObj:=wPaper;
    MoveL Offs(pOrigin,300.54,172.40,0.00),v40,z0,tPen\WObj:=wPaper;
    MoveL Offs(pOrigin,300.70,172.96,0.00),v40,z0,tPen\WObj:=wPaper;
    MoveL Offs(pOrigin,305.51,168.15,0.00),v40,z0,tPen\WObj:=wPaper;
    MoveL Offs(pOrigin,306.41,168.75,0.00),v40,z0,tPen\WObj:=wPaper;
    MoveL Offs(pOrigin,302.95,172.20,0.00),v40,z0,tPen\WObj:=wPaper;
    MoveL Offs(pOrigin,302.78,171.65,0.00),v40,z0,tPen\WObj:=wPaper;
    MoveL Offs(pOrigin,301.28,170.15,0.00),v40,z0,tPen\WObj:=wPaper;
    MoveL Offs(pOrigin,302.33,169.71,0.00),v40,z0,tPen\WObj:=wPaper;
    MoveL Offs(pOrigin,303.83,171.21,0.00),v40,fine,tPen\WObj:=wPaper;
    MoveL Offs(pOrigin,303.83,171.21,6.00),v60,z5,tPen\WObj:=wPaper;
    MoveL Offs(pOrigin,305.25,169.69,6.00),vTravel,z5,tPen\WObj:=wPaper;
    MoveL Offs(pOrigin,305.25,169.69,0.00),v60,z0,tPen\WObj:=wPaper;
    MoveL Offs(pOrigin,295.90,173.09,0.00),v40,z0,tPen\WObj:=wPaper;
    MoveL Offs(pOrigin,296.19,172.53,0.00),v40,z0,tPen\WObj:=wPaper;
    MoveL Offs(pOrigin,297.24,173.58,0.00),v40,z0,tPen\WObj:=wPaper;
    MoveL Offs(pOrigin,296.35,174.32,0.00),v40,z0,tPen\WObj:=wPaper;
    MoveL Offs(pOrigin,301.76,168.91,0.00),v40,fine,tPen\WObj:=wPaper;
    MoveL Offs(pOrigin,301.76,168.91,6.00),v60,z5,tPen\WObj:=wPaper;
    MoveL Offs(pOrigin,300.23,170.60,6.00),vTravel,z5,tPen\WObj:=wPaper;
    MoveL Offs(pOrigin,300.23,170.60,0.00),v60,z0,tPen\WObj:=wPaper;
    MoveL Offs(pOrigin,301.73,172.10,0.00),v40,fine,tPen\WObj:=wPaper;
    MoveL Offs(pOrigin,301.73,172.10,6.00),v60,z5,tPen\WObj:=wPaper;
    MoveL Offs(pOrigin,299.49,172.84,6.00),vTravel,z5,tPen\WObj:=wPaper;
    MoveL Offs(pOrigin,299.49,172.84,0.00),v60,z0,tPen\WObj:=wPaper;
    MoveL Offs(pOrigin,298.14,171.49,0.00),v40,fine,tPen\WObj:=wPaper;
    MoveL Offs(pOrigin,298.14,171.49,6.00),v60,z5,tPen\WObj:=wPaper;
    MoveL Offs(pOrigin,304.72,169.11,6.00),vTravel,z5,tPen\WObj:=wPaper;
    MoveL Offs(pOrigin,304.72,169.11,0.00),v60,z0,tPen\WObj:=wPaper;
    MoveL Offs(pOrigin,305.77,170.17,0.00),v40,fine,tPen\WObj:=wPaper;
    MoveL Offs(pOrigin,305.77,170.17,6.00),v60,z5,tPen\WObj:=wPaper;
    MoveL Offs(pOrigin,313.00,183.37,6.00),vTravel,z5,tPen\WObj:=wPaper;
    MoveL Offs(pOrigin,313.00,183.37,0.00),v60,z0,tPen\WObj:=wPaper;
    MoveL Offs(pOrigin,314.51,184.87,0.00),v40,fine,tPen\WObj:=wPaper;
    MoveL Offs(pOrigin,314.51,184.87,6.00),v60,z5,tPen\WObj:=wPaper;
    MoveL Offs(pOrigin,319.39,185.63,6.00),vTravel,z5,tPen\WObj:=wPaper;
    MoveL Offs(pOrigin,319.39,185.63,0.00),v60,z0,tPen\WObj:=wPaper;
    MoveL Offs(pOrigin,321.79,183.23,0.00),v40,fine,tPen\WObj:=wPaper;
    MoveL Offs(pOrigin,321.79,183.23,6.00),v60,z5,tPen\WObj:=wPaper;
    MoveL Offs(pOrigin,321.03,188.48,6.00),vTravel,z5,tPen\WObj:=wPaper;
    MoveL Offs(pOrigin,321.03,188.48,0.00),v60,z0,tPen\WObj:=wPaper;
  ENDPROC

  PROC DrawPart216()
    MoveL Offs(pOrigin,307.50,202.00,0.00),v40,fine,tPen\WObj:=wPaper;
    MoveL Offs(pOrigin,307.50,202.00,6.00),v60,z5,tPen\WObj:=wPaper;
    MoveL Offs(pOrigin,305.04,206.45,6.00),vTravel,z5,tPen\WObj:=wPaper;
    MoveL Offs(pOrigin,305.04,206.45,0.00),v60,z0,tPen\WObj:=wPaper;
    MoveL Offs(pOrigin,304.61,206.88,0.00),v40,z0,tPen\WObj:=wPaper;
    MoveL Offs(pOrigin,305.04,206.45,0.00),v40,z0,tPen\WObj:=wPaper;
    MoveL Offs(pOrigin,304.69,206.41,0.00),v40,z0,tPen\WObj:=wPaper;
    MoveL Offs(pOrigin,306.19,207.92,0.00),v40,z0,tPen\WObj:=wPaper;
    MoveL Offs(pOrigin,305.89,207.94,0.00),v40,z0,tPen\WObj:=wPaper;
    MoveL Offs(pOrigin,306.10,207.51,0.00),v40,z0,tPen\WObj:=wPaper;
    MoveL Offs(pOrigin,305.89,207.94,0.00),v40,fine,tPen\WObj:=wPaper;
    MoveL Offs(pOrigin,305.89,207.94,6.00),v60,z5,tPen\WObj:=wPaper;
    MoveL Offs(pOrigin,304.83,209.21,6.00),vTravel,z5,tPen\WObj:=wPaper;
    MoveL Offs(pOrigin,304.83,209.21,0.00),v60,z0,tPen\WObj:=wPaper;
    MoveL Offs(pOrigin,305.04,208.79,0.00),v40,z0,tPen\WObj:=wPaper;
    MoveL Offs(pOrigin,304.83,209.21,0.00),v40,fine,tPen\WObj:=wPaper;
    MoveL Offs(pOrigin,304.83,209.21,6.00),v60,z5,tPen\WObj:=wPaper;
    MoveL Offs(pOrigin,287.19,197.69,6.00),vTravel,z5,tPen\WObj:=wPaper;
    MoveL Offs(pOrigin,287.19,197.69,0.00),v60,z0,tPen\WObj:=wPaper;
    MoveL Offs(pOrigin,285.70,197.69,0.00),v40,z0,tPen\WObj:=wPaper;
    MoveL Offs(pOrigin,284.75,197.87,0.00),v40,z0,tPen\WObj:=wPaper;
    MoveL Offs(pOrigin,287.30,195.32,0.00),v40,z0,tPen\WObj:=wPaper;
    MoveL Offs(pOrigin,286.34,195.58,0.00),v40,z0,tPen\WObj:=wPaper;
    MoveL Offs(pOrigin,285.27,195.58,0.00),v40,z0,tPen\WObj:=wPaper;
    MoveL Offs(pOrigin,285.49,196.63,0.00),v40,z0,tPen\WObj:=wPaper;
    MoveL Offs(pOrigin,286.55,196.63,0.00),v40,fine,tPen\WObj:=wPaper;
    MoveL Offs(pOrigin,286.55,196.63,6.00),v60,z5,tPen\WObj:=wPaper;
    MoveL Offs(pOrigin,286.12,194.52,6.00),vTravel,z5,tPen\WObj:=wPaper;
    MoveL Offs(pOrigin,286.12,194.52,0.00),v60,z0,tPen\WObj:=wPaper;
    MoveL Offs(pOrigin,284.85,194.52,0.00),v40,z0,tPen\WObj:=wPaper;
    MoveL Offs(pOrigin,284.64,193.46,0.00),v40,z0,tPen\WObj:=wPaper;
    MoveL Offs(pOrigin,285.91,193.46,0.00),v40,z0,tPen\WObj:=wPaper;
    MoveL Offs(pOrigin,286.71,192.93,0.00),v40,z0,tPen\WObj:=wPaper;
    MoveL Offs(pOrigin,284.00,195.63,0.00),v40,fine,tPen\WObj:=wPaper;
    MoveL Offs(pOrigin,284.00,195.63,6.00),v60,z5,tPen\WObj:=wPaper;
    MoveL Offs(pOrigin,284.42,192.41,6.00),vTravel,z5,tPen\WObj:=wPaper;
    MoveL Offs(pOrigin,284.42,192.41,0.00),v60,z0,tPen\WObj:=wPaper;
    MoveL Offs(pOrigin,285.49,192.41,0.00),v40,fine,tPen\WObj:=wPaper;
    MoveL Offs(pOrigin,285.49,192.41,6.00),v60,z5,tPen\WObj:=wPaper;
    MoveL Offs(pOrigin,275.77,194.91,6.00),vTravel,z5,tPen\WObj:=wPaper;
    MoveL Offs(pOrigin,275.77,194.91,0.00),v60,z0,tPen\WObj:=wPaper;
    MoveL Offs(pOrigin,272.76,197.91,0.00),v40,fine,tPen\WObj:=wPaper;
    MoveL Offs(pOrigin,272.76,197.91,6.00),v60,z5,tPen\WObj:=wPaper;
    MoveL Offs(pOrigin,274.57,197.52,6.00),vTravel,z5,tPen\WObj:=wPaper;
    MoveL Offs(pOrigin,274.57,197.52,0.00),v60,z0,tPen\WObj:=wPaper;
    MoveL Offs(pOrigin,274.57,196.04,0.00),v40,z0,tPen\WObj:=wPaper;
    MoveL Offs(pOrigin,275.08,195.58,0.00),v40,z0,tPen\WObj:=wPaper;
    MoveL Offs(pOrigin,273.16,195.58,0.00),v40,z0,tPen\WObj:=wPaper;
    MoveL Offs(pOrigin,272.95,194.52,0.00),v40,z0,tPen\WObj:=wPaper;
    MoveL Offs(pOrigin,274.44,194.52,0.00),v40,z0,tPen\WObj:=wPaper;
    MoveL Offs(pOrigin,274.86,194.76,0.00),v40,z0,tPen\WObj:=wPaper;
    MoveL Offs(pOrigin,275.08,195.19,0.00),v40,z0,tPen\WObj:=wPaper;
    MoveL Offs(pOrigin,274.86,194.76,0.00),v40,fine,tPen\WObj:=wPaper;
    MoveL Offs(pOrigin,274.86,194.76,6.00),v60,z5,tPen\WObj:=wPaper;
    MoveL Offs(pOrigin,272.95,194.12,6.00),vTravel,z5,tPen\WObj:=wPaper;
    MoveL Offs(pOrigin,272.95,194.12,0.00),v60,z0,tPen\WObj:=wPaper;
    MoveL Offs(pOrigin,273.38,194.76,0.00),v40,z0,tPen\WObj:=wPaper;
    MoveL Offs(pOrigin,272.95,194.12,0.00),v40,fine,tPen\WObj:=wPaper;
    MoveL Offs(pOrigin,272.95,194.12,6.00),v60,z5,tPen\WObj:=wPaper;
    MoveL Offs(pOrigin,273.59,192.85,6.00),vTravel,z5,tPen\WObj:=wPaper;
    MoveL Offs(pOrigin,273.59,192.85,0.00),v60,z0,tPen\WObj:=wPaper;
    MoveL Offs(pOrigin,273.80,193.27,0.00),v40,z0,tPen\WObj:=wPaper;
    MoveL Offs(pOrigin,273.59,192.85,0.00),v40,z0,tPen\WObj:=wPaper;
    MoveL Offs(pOrigin,273.16,192.41,0.00),v40,z0,tPen\WObj:=wPaper;
    MoveL Offs(pOrigin,271.68,192.41,0.00),v40,fine,tPen\WObj:=wPaper;
    MoveL Offs(pOrigin,271.68,192.41,6.00),v60,z5,tPen\WObj:=wPaper;
    MoveL Offs(pOrigin,274.22,189.39,6.00),vTravel,z5,tPen\WObj:=wPaper;
    MoveL Offs(pOrigin,274.22,189.39,0.00),v60,z0,tPen\WObj:=wPaper;
    MoveL Offs(pOrigin,269.87,185.04,0.00),v40,z0,tPen\WObj:=wPaper;
    MoveL Offs(pOrigin,270.19,184.35,0.00),v40,z0,tPen\WObj:=wPaper;
    MoveL Offs(pOrigin,270.40,184.77,0.00),v40,z0,tPen\WObj:=wPaper;
    MoveL Offs(pOrigin,270.19,184.35,0.00),v40,fine,tPen\WObj:=wPaper;
    MoveL Offs(pOrigin,270.19,184.35,6.00),v60,z5,tPen\WObj:=wPaper;
    MoveL Offs(pOrigin,271.46,184.28,6.00),vTravel,z5,tPen\WObj:=wPaper;
    MoveL Offs(pOrigin,271.46,184.28,0.00),v60,z0,tPen\WObj:=wPaper;
    MoveL Offs(pOrigin,266.95,188.79,0.00),v40,z0,tPen\WObj:=wPaper;
    MoveL Offs(pOrigin,267.84,189.39,0.00),v40,z0,tPen\WObj:=wPaper;
    MoveL Offs(pOrigin,272.05,185.18,0.00),v40,fine,tPen\WObj:=wPaper;
    MoveL Offs(pOrigin,272.05,185.18,6.00),v60,z5,tPen\WObj:=wPaper;
    MoveL Offs(pOrigin,267.42,183.96,6.00),vTravel,z5,tPen\WObj:=wPaper;
    MoveL Offs(pOrigin,267.42,183.96,0.00),v60,z0,tPen\WObj:=wPaper;
    MoveL Offs(pOrigin,266.15,183.96,0.00),v40,fine,tPen\WObj:=wPaper;
    MoveL Offs(pOrigin,266.15,183.96,6.00),v60,z5,tPen\WObj:=wPaper;
    MoveL Offs(pOrigin,265.51,182.90,6.00),vTravel,z5,tPen\WObj:=wPaper;
    MoveL Offs(pOrigin,265.51,182.90,0.00),v60,z0,tPen\WObj:=wPaper;
    MoveL Offs(pOrigin,266.79,182.90,0.00),v40,fine,tPen\WObj:=wPaper;
    MoveL Offs(pOrigin,266.79,182.90,6.00),v60,z5,tPen\WObj:=wPaper;
    MoveL Offs(pOrigin,265.73,181.16,6.00),vTravel,z5,tPen\WObj:=wPaper;
    MoveL Offs(pOrigin,265.73,181.16,0.00),v60,z0,tPen\WObj:=wPaper;
    MoveL Offs(pOrigin,265.94,181.59,0.00),v40,z0,tPen\WObj:=wPaper;
    MoveL Offs(pOrigin,265.73,181.16,0.00),v40,fine,tPen\WObj:=wPaper;
    MoveL Offs(pOrigin,265.73,181.16,6.00),v60,z5,tPen\WObj:=wPaper;
    MoveL Offs(pOrigin,264.57,183.71,6.00),vTravel,z5,tPen\WObj:=wPaper;
    MoveL Offs(pOrigin,264.57,183.71,0.00),v60,z0,tPen\WObj:=wPaper;
    MoveL Offs(pOrigin,268.47,179.80,0.00),v40,fine,tPen\WObj:=wPaper;
    MoveL Offs(pOrigin,268.47,179.80,6.00),v60,z5,tPen\WObj:=wPaper;
    MoveL Offs(pOrigin,269.23,177.55,6.00),vTravel,z5,tPen\WObj:=wPaper;
    MoveL Offs(pOrigin,269.23,177.55,0.00),v60,z0,tPen\WObj:=wPaper;
    MoveL Offs(pOrigin,270.58,176.20,0.00),v40,z0,tPen\WObj:=wPaper;
    MoveL Offs(pOrigin,271.48,176.79,0.00),v40,z0,tPen\WObj:=wPaper;
    MoveL Offs(pOrigin,270.28,178.00,0.00),v40,z0,tPen\WObj:=wPaper;
    MoveL Offs(pOrigin,271.17,178.59,0.00),v40,z0,tPen\WObj:=wPaper;
    MoveL Offs(pOrigin,272.53,177.24,0.00),v40,z0,tPen\WObj:=wPaper;
    MoveL Offs(pOrigin,273.57,177.69,0.00),v40,z0,tPen\WObj:=wPaper;
    MoveL Offs(pOrigin,272.07,179.19,0.00),v40,z0,tPen\WObj:=wPaper;
    MoveL Offs(pOrigin,273.12,179.64,0.00),v40,z0,tPen\WObj:=wPaper;
    MoveL Offs(pOrigin,274.47,178.28,0.00),v40,z0,tPen\WObj:=wPaper;
    MoveL Offs(pOrigin,275.22,177.53,0.00),v40,z0,tPen\WObj:=wPaper;
    MoveL Offs(pOrigin,277.47,175.28,0.00),v40,z0,tPen\WObj:=wPaper;
    MoveL Offs(pOrigin,276.43,175.17,0.00),v40,z0,tPen\WObj:=wPaper;
    MoveL Offs(pOrigin,275.38,174.12,0.00),v40,fine,tPen\WObj:=wPaper;
    MoveL Offs(pOrigin,275.38,174.12,6.00),v60,z5,tPen\WObj:=wPaper;
    MoveL Offs(pOrigin,276.58,173.18,6.00),vTravel,z5,tPen\WObj:=wPaper;
    MoveL Offs(pOrigin,276.58,173.18,0.00),v60,z0,tPen\WObj:=wPaper;
    MoveL Offs(pOrigin,274.18,175.59,0.00),v40,z0,tPen\WObj:=wPaper;
    MoveL Offs(pOrigin,274.77,176.48,0.00),v40,z0,tPen\WObj:=wPaper;
    MoveL Offs(pOrigin,277.03,174.23,0.00),v40,fine,tPen\WObj:=wPaper;
    MoveL Offs(pOrigin,277.03,174.23,6.00),v60,z5,tPen\WObj:=wPaper;
    MoveL Offs(pOrigin,275.99,172.29,6.00),vTravel,z5,tPen\WObj:=wPaper;
    MoveL Offs(pOrigin,275.99,172.29,0.00),v60,z0,tPen\WObj:=wPaper;
  ENDPROC

  PROC DrawPart217()
    MoveL Offs(pOrigin,273.58,174.69,0.00),v40,z0,tPen\WObj:=wPaper;
    MoveL Offs(pOrigin,273.14,173.64,0.00),v40,z0,tPen\WObj:=wPaper;
    MoveL Offs(pOrigin,275.54,171.24,0.00),v40,z0,tPen\WObj:=wPaper;
    MoveL Offs(pOrigin,275.09,170.19,0.00),v40,z0,tPen\WObj:=wPaper;
    MoveL Offs(pOrigin,273.14,172.15,0.00),v40,fine,tPen\WObj:=wPaper;
    MoveL Offs(pOrigin,273.14,172.15,6.00),v60,z5,tPen\WObj:=wPaper;
    MoveL Offs(pOrigin,272.99,170.80,6.00),vTravel,z5,tPen\WObj:=wPaper;
    MoveL Offs(pOrigin,272.99,170.80,0.00),v60,z0,tPen\WObj:=wPaper;
    MoveL Offs(pOrigin,274.50,169.29,0.00),v40,z0,tPen\WObj:=wPaper;
    MoveL Offs(pOrigin,274.05,168.25,0.00),v40,z0,tPen\WObj:=wPaper;
    MoveL Offs(pOrigin,272.55,169.75,0.00),v40,z0,tPen\WObj:=wPaper;
    MoveL Offs(pOrigin,272.10,168.70,0.00),v40,z0,tPen\WObj:=wPaper;
    MoveL Offs(pOrigin,273.75,167.05,0.00),v40,z0,tPen\WObj:=wPaper;
    MoveL Offs(pOrigin,273.16,166.15,0.00),v40,z0,tPen\WObj:=wPaper;
    MoveL Offs(pOrigin,271.66,167.66,0.00),v40,fine,tPen\WObj:=wPaper;
    MoveL Offs(pOrigin,271.66,167.66,6.00),v60,z5,tPen\WObj:=wPaper;
    MoveL Offs(pOrigin,271.36,166.46,6.00),vTravel,z5,tPen\WObj:=wPaper;
    MoveL Offs(pOrigin,271.36,166.46,0.00),v60,z0,tPen\WObj:=wPaper;
    MoveL Offs(pOrigin,272.71,165.11,0.00),v40,z0,tPen\WObj:=wPaper;
    MoveL Offs(pOrigin,272.27,164.06,0.00),v40,z0,tPen\WObj:=wPaper;
    MoveL Offs(pOrigin,270.91,165.41,0.00),v40,z0,tPen\WObj:=wPaper;
    MoveL Offs(pOrigin,270.47,164.36,0.00),v40,z0,tPen\WObj:=wPaper;
    MoveL Offs(pOrigin,271.82,163.01,0.00),v40,z0,tPen\WObj:=wPaper;
    MoveL Offs(pOrigin,271.37,161.96,0.00),v40,z0,tPen\WObj:=wPaper;
    MoveL Offs(pOrigin,270.02,163.32,0.00),v40,fine,tPen\WObj:=wPaper;
    MoveL Offs(pOrigin,270.02,163.32,6.00),v60,z5,tPen\WObj:=wPaper;
    MoveL Offs(pOrigin,269.73,162.12,6.00),vTravel,z5,tPen\WObj:=wPaper;
    MoveL Offs(pOrigin,269.73,162.12,0.00),v60,z0,tPen\WObj:=wPaper;
    MoveL Offs(pOrigin,270.78,161.07,0.00),v40,z0,tPen\WObj:=wPaper;
    MoveL Offs(pOrigin,270.33,160.02,0.00),v40,z0,tPen\WObj:=wPaper;
    MoveL Offs(pOrigin,269.43,160.92,0.00),v40,fine,tPen\WObj:=wPaper;
    MoveL Offs(pOrigin,269.43,160.92,6.00),v60,z5,tPen\WObj:=wPaper;
    MoveL Offs(pOrigin,276.99,160.73,6.00),vTravel,z5,tPen\WObj:=wPaper;
    MoveL Offs(pOrigin,276.99,160.73,0.00),v60,z0,tPen\WObj:=wPaper;
    MoveL Offs(pOrigin,278.26,160.73,0.00),v40,fine,tPen\WObj:=wPaper;
    MoveL Offs(pOrigin,278.26,160.73,6.00),v60,z5,tPen\WObj:=wPaper;
    MoveL Offs(pOrigin,279.91,163.89,6.00),vTravel,z5,tPen\WObj:=wPaper;
    MoveL Offs(pOrigin,279.91,163.89,0.00),v60,z0,tPen\WObj:=wPaper;
    MoveL Offs(pOrigin,277.05,166.74,0.00),v40,fine,tPen\WObj:=wPaper;
    MoveL Offs(pOrigin,277.05,166.74,6.00),v60,z5,tPen\WObj:=wPaper;
    MoveL Offs(pOrigin,277.35,167.94,6.00),vTravel,z5,tPen\WObj:=wPaper;
    MoveL Offs(pOrigin,277.35,167.94,0.00),v60,z0,tPen\WObj:=wPaper;
    MoveL Offs(pOrigin,280.20,165.08,0.00),v40,fine,tPen\WObj:=wPaper;
    MoveL Offs(pOrigin,280.20,165.08,6.00),v60,z5,tPen\WObj:=wPaper;
    MoveL Offs(pOrigin,280.64,167.63,6.00),vTravel,z5,tPen\WObj:=wPaper;
    MoveL Offs(pOrigin,280.64,167.63,0.00),v60,z0,tPen\WObj:=wPaper;
    MoveL Offs(pOrigin,277.94,170.33,0.00),v40,fine,tPen\WObj:=wPaper;
    MoveL Offs(pOrigin,277.94,170.33,6.00),v60,z5,tPen\WObj:=wPaper;
    MoveL Offs(pOrigin,278.90,169.18,6.00),vTravel,z5,tPen\WObj:=wPaper;
    MoveL Offs(pOrigin,278.90,169.18,0.00),v60,z0,tPen\WObj:=wPaper;
    MoveL Offs(pOrigin,279.96,169.18,0.00),v40,z0,tPen\WObj:=wPaper;
    MoveL Offs(pOrigin,279.75,168.12,0.00),v40,z0,tPen\WObj:=wPaper;
    MoveL Offs(pOrigin,278.69,168.12,0.00),v40,fine,tPen\WObj:=wPaper;
    MoveL Offs(pOrigin,278.69,168.12,6.00),v60,z5,tPen\WObj:=wPaper;
    MoveL Offs(pOrigin,281.68,172.57,6.00),vTravel,z5,tPen\WObj:=wPaper;
    MoveL Offs(pOrigin,281.68,172.57,0.00),v60,z0,tPen\WObj:=wPaper;
    MoveL Offs(pOrigin,274.01,180.23,0.00),v40,z0,tPen\WObj:=wPaper;
    MoveL Offs(pOrigin,274.76,180.98,0.00),v40,z0,tPen\WObj:=wPaper;
    MoveL Offs(pOrigin,282.12,173.62,0.00),v40,fine,tPen\WObj:=wPaper;
    MoveL Offs(pOrigin,282.12,173.62,6.00),v60,z5,tPen\WObj:=wPaper;
    MoveL Offs(pOrigin,277.41,178.40,6.00),vTravel,z5,tPen\WObj:=wPaper;
    MoveL Offs(pOrigin,277.41,178.40,0.00),v60,z0,tPen\WObj:=wPaper;
    MoveL Offs(pOrigin,276.49,176.91,0.00),v40,z0,tPen\WObj:=wPaper;
    MoveL Offs(pOrigin,275.15,176.06,0.00),v40,z0,tPen\WObj:=wPaper;
    MoveL Offs(pOrigin,271.25,170.54,0.00),v40,fine,tPen\WObj:=wPaper;
    MoveL Offs(pOrigin,271.25,170.54,6.00),v60,z5,tPen\WObj:=wPaper;
    MoveL Offs(pOrigin,268.35,172.46,6.00),vTravel,z5,tPen\WObj:=wPaper;
    MoveL Offs(pOrigin,268.35,172.46,0.00),v60,z0,tPen\WObj:=wPaper;
    MoveL Offs(pOrigin,266.99,173.81,0.00),v40,z0,tPen\WObj:=wPaper;
    MoveL Offs(pOrigin,266.40,172.91,0.00),v40,z0,tPen\WObj:=wPaper;
    MoveL Offs(pOrigin,267.75,171.56,0.00),v40,z0,tPen\WObj:=wPaper;
    MoveL Offs(pOrigin,267.15,170.67,0.00),v40,z0,tPen\WObj:=wPaper;
    MoveL Offs(pOrigin,265.80,172.02,0.00),v40,fine,tPen\WObj:=wPaper;
    MoveL Offs(pOrigin,265.80,172.02,6.00),v60,z5,tPen\WObj:=wPaper;
    MoveL Offs(pOrigin,264.24,174.57,6.00),vTravel,z5,tPen\WObj:=wPaper;
    MoveL Offs(pOrigin,264.24,174.57,0.00),v60,z0,tPen\WObj:=wPaper;
    MoveL Offs(pOrigin,269.34,176.27,0.00),v40,z0,tPen\WObj:=wPaper;
    MoveL Offs(pOrigin,269.68,175.60,0.00),v40,z0,tPen\WObj:=wPaper;
    MoveL Offs(pOrigin,268.33,176.95,0.00),v40,z0,tPen\WObj:=wPaper;
    MoveL Offs(pOrigin,267.43,176.36,0.00),v40,z0,tPen\WObj:=wPaper;
    MoveL Offs(pOrigin,268.94,174.85,0.00),v40,fine,tPen\WObj:=wPaper;
    MoveL Offs(pOrigin,268.94,174.85,6.00),v60,z5,tPen\WObj:=wPaper;
    MoveL Offs(pOrigin,268.79,173.51,6.00),vTravel,z5,tPen\WObj:=wPaper;
    MoveL Offs(pOrigin,268.79,173.51,0.00),v60,z0,tPen\WObj:=wPaper;
    MoveL Offs(pOrigin,266.39,175.91,0.00),v40,fine,tPen\WObj:=wPaper;
    MoveL Offs(pOrigin,266.39,175.91,6.00),v60,z5,tPen\WObj:=wPaper;
    MoveL Offs(pOrigin,263.24,176.07,6.00),vTravel,z5,tPen\WObj:=wPaper;
    MoveL Offs(pOrigin,263.24,176.07,0.00),v60,z0,tPen\WObj:=wPaper;
    MoveL Offs(pOrigin,260.69,178.62,0.00),v40,z0,tPen\WObj:=wPaper;
    MoveL Offs(pOrigin,259.94,177.88,0.00),v40,z0,tPen\WObj:=wPaper;
    MoveL Offs(pOrigin,262.64,175.17,0.00),v40,z0,tPen\WObj:=wPaper;
    MoveL Offs(pOrigin,261.69,175.51,0.00),v40,z0,tPen\WObj:=wPaper;
    MoveL Offs(pOrigin,260.62,175.51,0.00),v40,z0,tPen\WObj:=wPaper;
    MoveL Offs(pOrigin,260.20,174.46,0.00),v40,z0,tPen\WObj:=wPaper;
    MoveL Offs(pOrigin,261.26,174.46,0.00),v40,fine,tPen\WObj:=wPaper;
    MoveL Offs(pOrigin,261.26,174.46,6.00),v60,z5,tPen\WObj:=wPaper;
    MoveL Offs(pOrigin,261.75,173.08,6.00),vTravel,z5,tPen\WObj:=wPaper;
    MoveL Offs(pOrigin,261.75,173.08,0.00),v60,z0,tPen\WObj:=wPaper;
    MoveL Offs(pOrigin,259.20,175.63,0.00),v40,fine,tPen\WObj:=wPaper;
    MoveL Offs(pOrigin,259.20,175.63,6.00),v60,z5,tPen\WObj:=wPaper;
    MoveL Offs(pOrigin,249.74,167.90,6.00),vTravel,z5,tPen\WObj:=wPaper;
    MoveL Offs(pOrigin,249.74,167.90,0.00),v60,z0,tPen\WObj:=wPaper;
    MoveL Offs(pOrigin,248.24,166.39,0.00),v40,fine,tPen\WObj:=wPaper;
    MoveL Offs(pOrigin,248.24,166.39,6.00),v60,z5,tPen\WObj:=wPaper;
    MoveL Offs(pOrigin,246.35,164.59,6.00),vTravel,z5,tPen\WObj:=wPaper;
    MoveL Offs(pOrigin,246.35,164.59,0.00),v60,z0,tPen\WObj:=wPaper;
    MoveL Offs(pOrigin,245.45,165.49,0.00),v40,fine,tPen\WObj:=wPaper;
    MoveL Offs(pOrigin,245.45,165.49,6.00),v60,z5,tPen\WObj:=wPaper;
    MoveL Offs(pOrigin,243.20,164.75,6.00),vTravel,z5,tPen\WObj:=wPaper;
    MoveL Offs(pOrigin,243.20,164.75,0.00),v60,z0,tPen\WObj:=wPaper;
    MoveL Offs(pOrigin,223.52,184.43,0.00),v40,z0,tPen\WObj:=wPaper;
    MoveL Offs(pOrigin,224.18,184.15,0.00),v40,z0,tPen\WObj:=wPaper;
    MoveL Offs(pOrigin,225.83,185.80,0.00),v40,z0,tPen\WObj:=wPaper;
    MoveL Offs(pOrigin,225.35,186.07,0.00),v40,z0,tPen\WObj:=wPaper;
    MoveL Offs(pOrigin,224.29,186.07,0.00),v40,z0,tPen\WObj:=wPaper;
    MoveL Offs(pOrigin,224.08,187.13,0.00),v40,z0,tPen\WObj:=wPaper;
    MoveL Offs(pOrigin,225.14,187.13,0.00),v40,fine,tPen\WObj:=wPaper;
    MoveL Offs(pOrigin,225.14,187.13,6.00),v60,z5,tPen\WObj:=wPaper;
    MoveL Offs(pOrigin,226.36,186.07,6.00),vTravel,z5,tPen\WObj:=wPaper;
    MoveL Offs(pOrigin,226.36,186.07,0.00),v60,z0,tPen\WObj:=wPaper;
  ENDPROC

  PROC DrawPart218()
    MoveL Offs(pOrigin,222.30,190.13,0.00),v40,fine,tPen\WObj:=wPaper;
    MoveL Offs(pOrigin,222.30,190.13,6.00),v60,z5,tPen\WObj:=wPaper;
    MoveL Offs(pOrigin,222.46,188.48,6.00),vTravel,z5,tPen\WObj:=wPaper;
    MoveL Offs(pOrigin,222.46,188.48,0.00),v60,z0,tPen\WObj:=wPaper;
    MoveL Offs(pOrigin,233.88,177.06,0.00),v40,z0,tPen\WObj:=wPaper;
    MoveL Offs(pOrigin,234.77,177.66,0.00),v40,z0,tPen\WObj:=wPaper;
    MoveL Offs(pOrigin,236.88,175.55,0.00),v40,fine,tPen\WObj:=wPaper;
    MoveL Offs(pOrigin,236.88,175.55,6.00),v60,z5,tPen\WObj:=wPaper;
    MoveL Offs(pOrigin,237.78,176.85,6.00),vTravel,z5,tPen\WObj:=wPaper;
    MoveL Offs(pOrigin,237.78,176.85,0.00),v60,z0,tPen\WObj:=wPaper;
    MoveL Offs(pOrigin,239.29,178.35,0.00),v40,fine,tPen\WObj:=wPaper;
    MoveL Offs(pOrigin,239.29,178.35,6.00),v60,z5,tPen\WObj:=wPaper;
    MoveL Offs(pOrigin,240.34,179.40,6.00),vTravel,z5,tPen\WObj:=wPaper;
    MoveL Offs(pOrigin,240.34,179.40,0.00),v60,z0,tPen\WObj:=wPaper;
    MoveL Offs(pOrigin,242.44,181.51,0.00),v40,z0,tPen\WObj:=wPaper;
    MoveL Offs(pOrigin,243.19,180.76,0.00),v40,z0,tPen\WObj:=wPaper;
    MoveL Offs(pOrigin,240.94,178.51,0.00),v40,z0,tPen\WObj:=wPaper;
    MoveL Offs(pOrigin,241.50,178.68,0.00),v40,z0,tPen\WObj:=wPaper;
    MoveL Offs(pOrigin,242.56,178.68,0.00),v40,z0,tPen\WObj:=wPaper;
    MoveL Offs(pOrigin,243.33,179.41,0.00),v40,z0,tPen\WObj:=wPaper;
    MoveL Offs(pOrigin,241.38,177.46,0.00),v40,z0,tPen\WObj:=wPaper;
    MoveL Offs(pOrigin,241.98,176.56,0.00),v40,z0,tPen\WObj:=wPaper;
    MoveL Offs(pOrigin,243.48,178.06,0.00),v40,z0,tPen\WObj:=wPaper;
    MoveL Offs(pOrigin,244.21,178.68,0.00),v40,z0,tPen\WObj:=wPaper;
    MoveL Offs(pOrigin,233.09,189.79,0.00),v40,fine,tPen\WObj:=wPaper;
    MoveL Offs(pOrigin,233.09,189.79,6.00),v60,z5,tPen\WObj:=wPaper;
    MoveL Offs(pOrigin,232.89,191.36,6.00),vTravel,z5,tPen\WObj:=wPaper;
    MoveL Offs(pOrigin,232.89,191.36,0.00),v60,z0,tPen\WObj:=wPaper;
    MoveL Offs(pOrigin,235.74,194.22,0.00),v40,z0,tPen\WObj:=wPaper;
    MoveL Offs(pOrigin,234.99,194.96,0.00),v40,z0,tPen\WObj:=wPaper;
    MoveL Offs(pOrigin,232.29,192.26,0.00),v40,z0,tPen\WObj:=wPaper;
    MoveL Offs(pOrigin,232.79,192.41,0.00),v40,z0,tPen\WObj:=wPaper;
    MoveL Offs(pOrigin,234.28,192.41,0.00),v40,z0,tPen\WObj:=wPaper;
    MoveL Offs(pOrigin,233.85,193.46,0.00),v40,z0,tPen\WObj:=wPaper;
    MoveL Offs(pOrigin,232.15,193.46,0.00),v40,z0,tPen\WObj:=wPaper;
    MoveL Offs(pOrigin,232.15,193.06,0.00),v40,z0,tPen\WObj:=wPaper;
    MoveL Offs(pOrigin,231.73,193.70,0.00),v40,z0,tPen\WObj:=wPaper;
    MoveL Offs(pOrigin,232.15,193.06,0.00),v40,z0,tPen\WObj:=wPaper;
    MoveL Offs(pOrigin,232.33,194.12,0.00),v40,z0,tPen\WObj:=wPaper;
    MoveL Offs(pOrigin,232.33,196.04,0.00),v40,fine,tPen\WObj:=wPaper;
    MoveL Offs(pOrigin,232.33,196.04,6.00),v60,z5,tPen\WObj:=wPaper;
    MoveL Offs(pOrigin,233.64,191.35,6.00),vTravel,z5,tPen\WObj:=wPaper;
    MoveL Offs(pOrigin,233.64,191.35,0.00),v60,z0,tPen\WObj:=wPaper;
    MoveL Offs(pOrigin,234.91,191.35,0.00),v40,z0,tPen\WObj:=wPaper;
    MoveL Offs(pOrigin,235.12,191.15,0.00),v40,z0,tPen\WObj:=wPaper;
    MoveL Offs(pOrigin,234.70,191.57,0.00),v40,z0,tPen\WObj:=wPaper;
    MoveL Offs(pOrigin,235.12,191.15,0.00),v40,fine,tPen\WObj:=wPaper;
    MoveL Offs(pOrigin,235.12,191.15,6.00),v60,z5,tPen\WObj:=wPaper;
    MoveL Offs(pOrigin,237.58,191.28,6.00),vTravel,z5,tPen\WObj:=wPaper;
    MoveL Offs(pOrigin,237.58,191.28,0.00),v60,z0,tPen\WObj:=wPaper;
    MoveL Offs(pOrigin,213.69,215.17,0.00),v40,z0,tPen\WObj:=wPaper;
    MoveL Offs(pOrigin,214.09,215.87,0.00),v40,z0,tPen\WObj:=wPaper;
    MoveL Offs(pOrigin,215.59,217.38,0.00),v40,fine,tPen\WObj:=wPaper;
    MoveL Offs(pOrigin,215.59,217.38,6.00),v60,z5,tPen\WObj:=wPaper;
    MoveL Offs(pOrigin,216.42,215.64,6.00),vTravel,z5,tPen\WObj:=wPaper;
    MoveL Offs(pOrigin,216.42,215.64,0.00),v60,z0,tPen\WObj:=wPaper;
    MoveL Offs(pOrigin,214.72,215.64,0.00),v40,fine,tPen\WObj:=wPaper;
    MoveL Offs(pOrigin,214.72,215.64,6.00),v60,z5,tPen\WObj:=wPaper;
    MoveL Offs(pOrigin,216.49,214.74,6.00),vTravel,z5,tPen\WObj:=wPaper;
    MoveL Offs(pOrigin,216.49,214.74,0.00),v60,z0,tPen\WObj:=wPaper;
    MoveL Offs(pOrigin,216.49,211.76,0.00),v40,fine,tPen\WObj:=wPaper;
    MoveL Offs(pOrigin,216.49,211.76,6.00),v60,z5,tPen\WObj:=wPaper;
    MoveL Offs(pOrigin,217.55,212.40,6.00),vTravel,z5,tPen\WObj:=wPaper;
    MoveL Offs(pOrigin,217.55,212.40,0.00),v60,z0,tPen\WObj:=wPaper;
    MoveL Offs(pOrigin,217.55,214.10,0.00),v40,z0,tPen\WObj:=wPaper;
    MoveL Offs(pOrigin,217.83,215.14,0.00),v40,z0,tPen\WObj:=wPaper;
    MoveL Offs(pOrigin,213.47,210.78,0.00),v40,z0,tPen\WObj:=wPaper;
    MoveL Offs(pOrigin,214.09,210.36,0.00),v40,z0,tPen\WObj:=wPaper;
    MoveL Offs(pOrigin,215.79,210.36,0.00),v40,z0,tPen\WObj:=wPaper;
    MoveL Offs(pOrigin,216.40,209.47,0.00),v40,z0,tPen\WObj:=wPaper;
    MoveL Offs(pOrigin,211.89,213.98,0.00),v40,z0,tPen\WObj:=wPaper;
    MoveL Offs(pOrigin,211.98,213.77,0.00),v40,z0,tPen\WObj:=wPaper;
    MoveL Offs(pOrigin,209.28,211.06,0.00),v40,z0,tPen\WObj:=wPaper;
    MoveL Offs(pOrigin,209.36,210.54,0.00),v40,z0,tPen\WObj:=wPaper;
    MoveL Offs(pOrigin,206.65,213.24,0.00),v40,z0,tPen\WObj:=wPaper;
    MoveL Offs(pOrigin,206.74,213.00,0.00),v40,z0,tPen\WObj:=wPaper;
    MoveL Offs(pOrigin,203.73,210.00,0.00),v40,z0,tPen\WObj:=wPaper;
    MoveL Offs(pOrigin,204.42,209.51,0.00),v40,z0,tPen\WObj:=wPaper;
    MoveL Offs(pOrigin,202.01,211.91,0.00),v40,z0,tPen\WObj:=wPaper;
    MoveL Offs(pOrigin,200.97,211.46,0.00),v40,z0,tPen\WObj:=wPaper;
    MoveL Offs(pOrigin,203.37,209.06,0.00),v40,fine,tPen\WObj:=wPaper;
    MoveL Offs(pOrigin,203.37,209.06,6.00),v60,z5,tPen\WObj:=wPaper;
    MoveL Offs(pOrigin,201.34,209.30,6.00),vTravel,z5,tPen\WObj:=wPaper;
    MoveL Offs(pOrigin,201.34,209.30,0.00),v60,z0,tPen\WObj:=wPaper;
    MoveL Offs(pOrigin,197.94,209.30,0.00),v40,fine,tPen\WObj:=wPaper;
    MoveL Offs(pOrigin,197.94,209.30,6.00),v60,z5,tPen\WObj:=wPaper;
    MoveL Offs(pOrigin,196.63,209.83,6.00),vTravel,z5,tPen\WObj:=wPaper;
    MoveL Offs(pOrigin,196.63,209.83,0.00),v60,z0,tPen\WObj:=wPaper;
    MoveL Offs(pOrigin,199.03,207.43,0.00),v40,fine,tPen\WObj:=wPaper;
    MoveL Offs(pOrigin,199.03,207.43,6.00),v60,z5,tPen\WObj:=wPaper;
    MoveL Offs(pOrigin,198.59,203.38,6.00),vTravel,z5,tPen\WObj:=wPaper;
    MoveL Offs(pOrigin,198.59,203.38,0.00),v60,z0,tPen\WObj:=wPaper;
    MoveL Offs(pOrigin,193.64,208.34,0.00),v40,fine,tPen\WObj:=wPaper;
    MoveL Offs(pOrigin,193.64,208.34,6.00),v60,z5,tPen\WObj:=wPaper;
    MoveL Offs(pOrigin,203.46,211.42,6.00),vTravel,z5,tPen\WObj:=wPaper;
    MoveL Offs(pOrigin,203.46,211.42,0.00),v60,z0,tPen\WObj:=wPaper;
    MoveL Offs(pOrigin,209.84,211.42,0.00),v40,fine,tPen\WObj:=wPaper;
    MoveL Offs(pOrigin,209.84,211.42,6.00),v60,z5,tPen\WObj:=wPaper;
    MoveL Offs(pOrigin,207.78,211.06,6.00),vTravel,z5,tPen\WObj:=wPaper;
    MoveL Offs(pOrigin,207.78,211.06,0.00),v60,z0,tPen\WObj:=wPaper;
    MoveL Offs(pOrigin,210.33,213.61,0.00),v40,z0,tPen\WObj:=wPaper;
    MoveL Offs(pOrigin,210.55,213.83,0.00),v40,z0,tPen\WObj:=wPaper;
    MoveL Offs(pOrigin,215.50,208.87,0.00),v40,z0,tPen\WObj:=wPaper;
    MoveL Offs(pOrigin,214.94,209.30,0.00),v40,z0,tPen\WObj:=wPaper;
    MoveL Offs(pOrigin,213.02,209.30,0.00),v40,z0,tPen\WObj:=wPaper;
    MoveL Offs(pOrigin,212.12,209.43,0.00),v40,z0,tPen\WObj:=wPaper;
    MoveL Offs(pOrigin,207.91,205.22,0.00),v40,fine,tPen\WObj:=wPaper;
    MoveL Offs(pOrigin,207.91,205.22,6.00),v60,z5,tPen\WObj:=wPaper;
    MoveL Offs(pOrigin,206.98,203.96,6.00),vTravel,z5,tPen\WObj:=wPaper;
    MoveL Offs(pOrigin,206.98,203.96,0.00),v60,z0,tPen\WObj:=wPaper;
    MoveL Offs(pOrigin,209.23,201.70,0.00),v40,z0,tPen\WObj:=wPaper;
    MoveL Offs(pOrigin,208.77,202.41,0.00),v40,z0,tPen\WObj:=wPaper;
    MoveL Offs(pOrigin,209.84,203.48,0.00),v40,z0,tPen\WObj:=wPaper;
    MoveL Offs(pOrigin,208.77,202.41,0.00),v40,z0,tPen\WObj:=wPaper;
    MoveL Offs(pOrigin,209.20,202.97,0.00),v40,z0,tPen\WObj:=wPaper;
    MoveL Offs(pOrigin,207.50,202.97,0.00),v40,z0,tPen\WObj:=wPaper;
    MoveL Offs(pOrigin,207.07,202.84,0.00),v40,z0,tPen\WObj:=wPaper;
    MoveL Offs(pOrigin,207.93,203.69,0.00),v40,z0,tPen\WObj:=wPaper;
    MoveL Offs(pOrigin,207.07,202.84,0.00),v40,z0,tPen\WObj:=wPaper;
    MoveL Offs(pOrigin,206.38,203.06,0.00),v40,z0,tPen\WObj:=wPaper;
  ENDPROC

  PROC DrawPart219()
    MoveL Offs(pOrigin,208.49,200.96,0.00),v40,z0,tPen\WObj:=wPaper;
    MoveL Offs(pOrigin,207.93,201.35,0.00),v40,z0,tPen\WObj:=wPaper;
    MoveL Offs(pOrigin,208.35,201.77,0.00),v40,z0,tPen\WObj:=wPaper;
    MoveL Offs(pOrigin,207.93,201.35,0.00),v40,z0,tPen\WObj:=wPaper;
    MoveL Offs(pOrigin,208.14,201.91,0.00),v40,z0,tPen\WObj:=wPaper;
    MoveL Offs(pOrigin,206.65,201.91,0.00),v40,z0,tPen\WObj:=wPaper;
    MoveL Offs(pOrigin,206.44,201.99,0.00),v40,z0,tPen\WObj:=wPaper;
    MoveL Offs(pOrigin,206.86,202.41,0.00),v40,z0,tPen\WObj:=wPaper;
    MoveL Offs(pOrigin,206.44,201.99,0.00),v40,z0,tPen\WObj:=wPaper;
    MoveL Offs(pOrigin,205.79,202.16,0.00),v40,z0,tPen\WObj:=wPaper;
    MoveL Offs(pOrigin,207.89,200.06,0.00),v40,fine,tPen\WObj:=wPaper;
    MoveL Offs(pOrigin,207.89,200.06,6.00),v60,z5,tPen\WObj:=wPaper;
    MoveL Offs(pOrigin,209.83,202.60,6.00),vTravel,z5,tPen\WObj:=wPaper;
    MoveL Offs(pOrigin,209.83,202.60,0.00),v60,z0,tPen\WObj:=wPaper;
    MoveL Offs(pOrigin,205.02,207.41,0.00),v40,fine,tPen\WObj:=wPaper;
    MoveL Offs(pOrigin,205.02,207.41,6.00),v60,z5,tPen\WObj:=wPaper;
    MoveL Offs(pOrigin,206.37,207.55,6.00),vTravel,z5,tPen\WObj:=wPaper;
    MoveL Offs(pOrigin,206.37,207.55,0.00),v60,z0,tPen\WObj:=wPaper;
    MoveL Offs(pOrigin,210.58,203.35,0.00),v40,fine,tPen\WObj:=wPaper;
    MoveL Offs(pOrigin,210.58,203.35,6.00),v60,z5,tPen\WObj:=wPaper;
    MoveL Offs(pOrigin,210.16,205.18,6.00),vTravel,z5,tPen\WObj:=wPaper;
    MoveL Offs(pOrigin,210.16,205.18,0.00),v60,z0,tPen\WObj:=wPaper;
    MoveL Offs(pOrigin,210.16,207.30,0.00),v40,fine,tPen\WObj:=wPaper;
    MoveL Offs(pOrigin,210.16,207.30,6.00),v60,z5,tPen\WObj:=wPaper;
    MoveL Offs(pOrigin,209.81,208.59,6.00),vTravel,z5,tPen\WObj:=wPaper;
    MoveL Offs(pOrigin,209.81,208.59,0.00),v60,z0,tPen\WObj:=wPaper;
    MoveL Offs(pOrigin,212.67,205.74,0.00),v40,z0,tPen\WObj:=wPaper;
    MoveL Offs(pOrigin,213.41,206.48,0.00),v40,z0,tPen\WObj:=wPaper;
    MoveL Offs(pOrigin,210.86,209.04,0.00),v40,z0,tPen\WObj:=wPaper;
    MoveL Offs(pOrigin,211.76,209.63,0.00),v40,z0,tPen\WObj:=wPaper;
    MoveL Offs(pOrigin,214.16,207.23,0.00),v40,z0,tPen\WObj:=wPaper;
    MoveL Offs(pOrigin,213.02,207.19,0.00),v40,z0,tPen\WObj:=wPaper;
    MoveL Offs(pOrigin,208.78,207.19,0.00),v40,fine,tPen\WObj:=wPaper;
    MoveL Offs(pOrigin,208.78,207.19,6.00),v60,z5,tPen\WObj:=wPaper;
    MoveL Offs(pOrigin,208.01,210.39,6.00),vTravel,z5,tPen\WObj:=wPaper;
    MoveL Offs(pOrigin,208.01,210.39,0.00),v60,z0,tPen\WObj:=wPaper;
    MoveL Offs(pOrigin,205.46,212.95,0.00),v40,fine,tPen\WObj:=wPaper;
    MoveL Offs(pOrigin,205.46,212.95,6.00),v60,z5,tPen\WObj:=wPaper;
    MoveL Offs(pOrigin,212.72,211.52,6.00),vTravel,z5,tPen\WObj:=wPaper;
    MoveL Offs(pOrigin,212.72,211.52,0.00),v60,z0,tPen\WObj:=wPaper;
    MoveL Offs(pOrigin,217.08,215.88,0.00),v40,z0,tPen\WObj:=wPaper;
    MoveL Offs(pOrigin,216.85,215.38,0.00),v40,z0,tPen\WObj:=wPaper;
    MoveL Offs(pOrigin,214.94,217.29,0.00),v40,z0,tPen\WObj:=wPaper;
    MoveL Offs(pOrigin,216.85,215.38,0.00),v40,fine,tPen\WObj:=wPaper;
    MoveL Offs(pOrigin,216.85,215.38,6.00),v60,z5,tPen\WObj:=wPaper;
    MoveL Offs(pOrigin,219.66,212.40,6.00),vTravel,z5,tPen\WObj:=wPaper;
    MoveL Offs(pOrigin,219.66,212.40,0.00),v60,z0,tPen\WObj:=wPaper;
    MoveL Offs(pOrigin,219.66,210.70,0.00),v40,z0,tPen\WObj:=wPaper;
    MoveL Offs(pOrigin,219.19,211.12,0.00),v40,z0,tPen\WObj:=wPaper;
    MoveL Offs(pOrigin,218.98,211.55,0.00),v40,z0,tPen\WObj:=wPaper;
    MoveL Offs(pOrigin,219.19,211.12,0.00),v40,z0,tPen\WObj:=wPaper;
    MoveL Offs(pOrigin,218.98,211.42,0.00),v40,z0,tPen\WObj:=wPaper;
    MoveL Offs(pOrigin,221.52,211.42,0.00),v40,z0,tPen\WObj:=wPaper;
    MoveL Offs(pOrigin,222.01,211.85,0.00),v40,z0,tPen\WObj:=wPaper;
    MoveL Offs(pOrigin,219.31,209.15,0.00),v40,z0,tPen\WObj:=wPaper;
    MoveL Offs(pOrigin,219.61,209.30,0.00),v40,z0,tPen\WObj:=wPaper;
    MoveL Offs(pOrigin,222.59,209.30,0.00),v40,fine,tPen\WObj:=wPaper;
    MoveL Offs(pOrigin,222.59,209.30,6.00),v60,z5,tPen\WObj:=wPaper;
    MoveL Offs(pOrigin,223.66,210.51,6.00),vTravel,z5,tPen\WObj:=wPaper;
    MoveL Offs(pOrigin,223.66,210.51,0.00),v60,z0,tPen\WObj:=wPaper;
    MoveL Offs(pOrigin,219.60,206.45,0.00),v40,z0,tPen\WObj:=wPaper;
    MoveL Offs(pOrigin,219.11,206.76,0.00),v40,z0,tPen\WObj:=wPaper;
    MoveL Offs(pOrigin,222.71,203.16,0.00),v40,z0,tPen\WObj:=wPaper;
    MoveL Offs(pOrigin,222.29,203.16,0.00),v40,z0,tPen\WObj:=wPaper;
    MoveL Offs(pOrigin,220.33,201.21,0.00),v40,z0,tPen\WObj:=wPaper;
    MoveL Offs(pOrigin,219.72,201.67,0.00),v40,z0,tPen\WObj:=wPaper;
    MoveL Offs(pOrigin,223.78,197.61,0.00),v40,fine,tPen\WObj:=wPaper;
    MoveL Offs(pOrigin,223.78,197.61,6.00),v60,z5,tPen\WObj:=wPaper;
    MoveL Offs(pOrigin,222.59,198.74,6.00),vTravel,z5,tPen\WObj:=wPaper;
    MoveL Offs(pOrigin,222.59,198.74,0.00),v60,z0,tPen\WObj:=wPaper;
    MoveL Offs(pOrigin,221.52,198.74,0.00),v40,z0,tPen\WObj:=wPaper;
    MoveL Offs(pOrigin,220.92,198.82,0.00),v40,z0,tPen\WObj:=wPaper;
    MoveL Offs(pOrigin,222.73,200.62,0.00),v40,z0,tPen\WObj:=wPaper;
    MoveL Offs(pOrigin,222.16,200.86,0.00),v40,z0,tPen\WObj:=wPaper;
    MoveL Offs(pOrigin,221.10,200.86,0.00),v40,z0,tPen\WObj:=wPaper;
    MoveL Offs(pOrigin,220.63,200.01,0.00),v40,z0,tPen\WObj:=wPaper;
    MoveL Offs(pOrigin,222.58,201.97,0.00),v40,z0,tPen\WObj:=wPaper;
    MoveL Offs(pOrigin,221.95,201.91,0.00),v40,z0,tPen\WObj:=wPaper;
    MoveL Offs(pOrigin,220.89,201.91,0.00),v40,z0,tPen\WObj:=wPaper;
    MoveL Offs(pOrigin,220.19,202.56,0.00),v40,z0,tPen\WObj:=wPaper;
    MoveL Offs(pOrigin,221.99,204.36,0.00),v40,z0,tPen\WObj:=wPaper;
    MoveL Offs(pOrigin,221.52,204.02,0.00),v40,z0,tPen\WObj:=wPaper;
    MoveL Offs(pOrigin,220.46,204.02,0.00),v40,z0,tPen\WObj:=wPaper;
    MoveL Offs(pOrigin,220.68,202.97,0.00),v40,z0,tPen\WObj:=wPaper;
    MoveL Offs(pOrigin,221.74,202.97,0.00),v40,fine,tPen\WObj:=wPaper;
    MoveL Offs(pOrigin,221.74,202.97,6.00),v60,z5,tPen\WObj:=wPaper;
    MoveL Offs(pOrigin,222.56,204.81,6.00),vTravel,z5,tPen\WObj:=wPaper;
    MoveL Offs(pOrigin,222.56,204.81,0.00),v60,z0,tPen\WObj:=wPaper;
    MoveL Offs(pOrigin,218.65,208.71,0.00),v40,fine,tPen\WObj:=wPaper;
    MoveL Offs(pOrigin,218.65,208.71,6.00),v60,z5,tPen\WObj:=wPaper;
    MoveL Offs(pOrigin,220.04,207.19,6.00),vTravel,z5,tPen\WObj:=wPaper;
    MoveL Offs(pOrigin,220.04,207.19,0.00),v60,z0,tPen\WObj:=wPaper;
    MoveL Offs(pOrigin,221.31,207.19,0.00),v40,fine,tPen\WObj:=wPaper;
    MoveL Offs(pOrigin,221.31,207.19,6.00),v60,z5,tPen\WObj:=wPaper;
    MoveL Offs(pOrigin,220.72,208.58,6.00),vTravel,z5,tPen\WObj:=wPaper;
    MoveL Offs(pOrigin,220.72,208.58,0.00),v60,z0,tPen\WObj:=wPaper;
    MoveL Offs(pOrigin,220.72,211.34,0.00),v40,fine,tPen\WObj:=wPaper;
    MoveL Offs(pOrigin,220.72,211.34,6.00),v60,z5,tPen\WObj:=wPaper;
    MoveL Offs(pOrigin,220.52,213.35,6.00),vTravel,z5,tPen\WObj:=wPaper;
    MoveL Offs(pOrigin,220.52,213.35,0.00),v60,z0,tPen\WObj:=wPaper;
    MoveL Offs(pOrigin,218.42,211.24,0.00),v40,fine,tPen\WObj:=wPaper;
    MoveL Offs(pOrigin,218.42,211.24,6.00),v60,z5,tPen\WObj:=wPaper;
    MoveL Offs(pOrigin,223.01,207.19,6.00),vTravel,z5,tPen\WObj:=wPaper;
    MoveL Offs(pOrigin,223.01,207.19,0.00),v60,z0,tPen\WObj:=wPaper;
    MoveL Offs(pOrigin,224.50,207.19,0.00),v40,z0,tPen\WObj:=wPaper;
    MoveL Offs(pOrigin,225.00,207.37,0.00),v40,z0,tPen\WObj:=wPaper;
    MoveL Offs(pOrigin,223.49,205.86,0.00),v40,z0,tPen\WObj:=wPaper;
    MoveL Offs(pOrigin,224.08,206.14,0.00),v40,z0,tPen\WObj:=wPaper;
    MoveL Offs(pOrigin,225.56,206.14,0.00),v40,z0,tPen\WObj:=wPaper;
    MoveL Offs(pOrigin,225.74,206.62,0.00),v40,z0,tPen\WObj:=wPaper;
    MoveL Offs(pOrigin,224.39,205.27,0.00),v40,z0,tPen\WObj:=wPaper;
    MoveL Offs(pOrigin,224.43,205.74,0.00),v40,z0,tPen\WObj:=wPaper;
    MoveL Offs(pOrigin,222.16,207.94,0.00),v40,z0,tPen\WObj:=wPaper;
    MoveL Offs(pOrigin,224.43,205.74,0.00),v40,fine,tPen\WObj:=wPaper;
    MoveL Offs(pOrigin,224.43,205.74,6.00),v60,z5,tPen\WObj:=wPaper;
    MoveL Offs(pOrigin,222.90,206.76,6.00),vTravel,z5,tPen\WObj:=wPaper;
    MoveL Offs(pOrigin,222.90,206.76,0.00),v60,z0,tPen\WObj:=wPaper;
    MoveL Offs(pOrigin,224.40,208.26,0.00),v40,fine,tPen\WObj:=wPaper;
    MoveL Offs(pOrigin,224.40,208.26,6.00),v60,z5,tPen\WObj:=wPaper;
    MoveL Offs(pOrigin,226.14,210.19,6.00),vTravel,z5,tPen\WObj:=wPaper;
  ENDPROC

